// TIA Portal project "Fahrstuhl_V17" (V17)

(* hardware
DEVICE "S71500/ET200MP-Station_1"  S7-1500 station
   slot 0: "Profilschiene_0"  Rack  6ES7 590-1***0-0AA0
   slot 1: "SPS_Fahrstuhl"  CPU 1516F-3 PN/DP  6ES7 516-3FN01-0AB0  V2.9
      slot 3: "CPU-Display_1"  6ES7591-1BA00-0AA0
      slot 32768: "PROFINET-Schnittstelle_1"  X1
         slot 32769: "Port_1"  X1 P1
         slot 32770: "Port_2"  X1 P2
      slot 33024: "PROFINET-Schnittstelle_2"  X2
         slot 33025: "Port_1"  X2 P1
      slot 33280: "DP-Schnittstelle_1"  X3
      slot 34817: "Virtual CP interface port_1"  Virtual CP interface port  Virtual CP interface port
   slot 2: "DI 32x24VDC HF_1"  DI 32x24VDC HF  6ES7 521-1BL00-0AB0  V2.1
   slot 3: "DQ 32x24VDC/0.5A ST_1"  DQ 32x24VDC/0.5A ST  6ES7 522-1BL00-0AB0  V2.0
*)

// ===== PLC "SPS_Fahrstuhl"  CPU 1516F-3 PN/DP =====

VAR_GLOBAL   // PLC tag table "Standard-Variablentabelle"
   "Not-Aus" AT %I0.0 : Bool;   // Notausschalter Öffner
   "Automatikbetrieb" AT %I0.1 : Bool;   // Schalter Automatikbetrieb
   "Hand Hub Heben" AT %I0.2 : Bool;   // Schalter Kabine heben
   "Hand Hub Senken" AT %I0.3 : Bool;   // Schalter Kabine senken
   "Hand Tür auf" AT %I0.4 : Bool;   // Schalter Tür auf
   "Hand Tür zu" AT %I0.5 : Bool;   // Schalter Tür zu
   "Reserve_Eingang_0" AT %I0.6 : Bool;   // Reserve
   "Reserve_Eingang_1" AT %I0.7 : Bool;   // Reserve
   "Endlage zu tief" AT %I1.0 : Bool;   // Öffner
   "Endlage Etage I Halt" AT %I1.1 : Bool;   // Endlagenschalter Etage I Halt
   "Endlage Etage I Langsam" AT %I1.2 : Bool;   // Endlagenschalter Etage I Langsam
   "Endlage Etage II Halt" AT %I1.3 : Bool;   // Endlagenschalter Etage II Halt
   "Endlage Etage II Langsam" AT %I1.4 : Bool;   // Endlagenschalter Etage II Langsam
   "Endlage Etage III Halt" AT %I1.5 : Bool;   // Endlagenschalter Etage III Halt
   "Endlage Etage III Langsam" AT %I1.6 : Bool;   // Endlagenschalter Etage III Langsam
   "Endlage zu hoch" AT %I1.7 : Bool;   // Endlagenschalter zu hoch
   "Reserve_Eingang_2" AT %I2.0 : Bool;   // Reserve
   "Reserve_Eingang_3" AT %I2.1 : Bool;   // Reserve
   "Endlage Tür III Zu" AT %I2.2 : Bool;   // Endlagenschalter Tür III Zu
   "Endlage Tür III Auf" AT %I2.3 : Bool;   // Endlagenschalter Tür III Auf
   "Endlage Tür II Zu" AT %I2.4 : Bool;   // Endlagenschalter Tür II Zu
   "Endlage Tür II Auf" AT %I2.5 : Bool;   // Endlagenschalter Tür II Auf
   "Endlage Tür I Zu" AT %I2.6 : Bool;   // Endlagenschalter Tür I Zu
   "Endlage Tür I Auf" AT %I2.7 : Bool;   // Endlagenschalter Tür I Auf
   "Taster auf Etage III - Ab" AT %I3.0 : Bool;   // Taster auf Etage III - Ab
   "Taster auf Etage II - Ab" AT %I3.1 : Bool;   // Taster auf Etage II - Ab
   "Taster auf Etage II - Auf" AT %I3.2 : Bool;   // Taster auf Etage II - Auf
   "Taster auf Etage I - Auf" AT %I3.3 : Bool;   // Taster auf Etage I - Auf
   "Taster Lift nach III" AT %I3.4 : Bool;   // Taster Lift nach III
   "Taster Lift nach II" AT %I3.5 : Bool;   // Taster Lift nach II
   "Taster Lift nach I" AT %I3.6 : Bool;   // Taster Lift nach I
   "Reserve_Eingang_4" AT %I3.7 : Bool;   // Reserve
   "Hubmotor langsam Heben" AT %Q4.0 : Bool;   // Hubmotor langsam Heben
   "Hubmotor langsam Senken" AT %Q4.1 : Bool;   // Hubmotor langsam Senken
   "Hubmotor schnell Heben" AT %Q4.2 : Bool;   // Hubmotor schnell Heben
   "Hubmotor schnell Senken" AT %Q4.3 : Bool;   // Hubmotor schnell Senken
   "Türantrieb Etage I Öffnen" AT %Q4.4 : Bool;   // Türantrieb Etage I Öffnen
   "Türantrieb Etage I Schließen" AT %Q4.5 : Bool;   // Türantrieb Etage I Schließen
   "Türantrieb Etage II Öffnen" AT %Q4.6 : Bool;   // Türantrieb Etage II Öffnen
   "Türantrieb Etage II Schließen" AT %Q4.7 : Bool;   // Türantrieb Etage II Schließen
   "Türantrieb Etage III Öffnen" AT %Q5.0 : Bool;   // Türantrieb Etage III Öffnen
   "Türantrieb Etage III Schließen" AT %Q5.1 : Bool;   // Türantrieb Etage III Schließen
   "LED Lift nach I" AT %Q5.2 : Bool;   // LED Lift nach I
   "LED Lift nach II" AT %Q5.3 : Bool;   // LED Lift nach II
   "LED Lift nach III" AT %Q5.4 : Bool;   // LED Lift nach III
   "LED Etage I Lift Auf" AT %Q5.5 : Bool;   // LED Etage I Lift Auf
   "LED Etage II Lift Auf" AT %Q5.6 : Bool;   // LED Etage II Lift Auf
   "LED Etage II Lift Ab" AT %Q5.7 : Bool;   // LED Etage II Lift Ab
   "7-Segment G" AT %Q6.0 : Bool;   // 7-Segment G
   "7-Segment A" AT %Q6.1 : Bool;   // 7-Segment A
   "7-Segment B" AT %Q6.2 : Bool;   // 7-Segment B
   "7-Segment C" AT %Q6.3 : Bool;   // 7-Segment C
   "7-Segment D" AT %Q6.4 : Bool;   // 7-Segment D
   "7-Segment E" AT %Q6.5 : Bool;   // 7-Segment E
   "7-Segment F" AT %Q6.6 : Bool;   // 7-Segment F
   "LED Etage Lift III Ab" AT %Q6.7 : Bool;   // LED Etage Lift III Ab
   "Reserve_Ausgang_0" AT %Q7.0 : Bool;   // Reserve
   "Reserve_Ausgang_1" AT %Q7.1 : Bool;   // Reserve
   "Reserve_Ausgang_2" AT %Q7.2 : Bool;   // Reserve
   "Reserve_Ausgang_3" AT %Q7.3 : Bool;   // Reserve
   "Reserve_Ausgang_4" AT %Q7.4 : Bool;   // Reserve
   "Reserve_Ausgang_5" AT %Q7.5 : Bool;   // Reserve
   "Reserve_Ausgang_6" AT %Q7.6 : Bool;   // Reserve
   "Reserve_Ausgang_7" AT %Q7.7 : Bool;   // Reserve
   "Clock_Byte" AT %MB0 : Byte;
   "Clock_10Hz" AT %M0.0 : Bool;
   "Clock_5Hz" AT %M0.1 : Bool;
   "Clock_2.5Hz" AT %M0.2 : Bool;
   "Clock_2Hz" AT %M0.3 : Bool;
   "Clock_1.25Hz" AT %M0.4 : Bool;
   "Clock_1Hz" AT %M0.5 : Bool;
   "Clock_0.625Hz" AT %M0.6 : Bool;
   "Clock_0.5Hz" AT %M0.7 : Bool;
END_VAR

// folder: IDB's

DATA_BLOCK "Tür zu_DB"   // DB1
{ S7_Optimized_Access := 'TRUE' }
VERSION : 0.1
// stored: InstanceOfName Tür zu
"Tür zu"
BEGIN
END_DATA_BLOCK

DATA_BLOCK "Tür auf_DB"   // DB2
{ S7_Optimized_Access := 'TRUE' }
VERSION : 0.1
// stored: InstanceOfName Tür auf
"Tür auf"
BEGIN
END_DATA_BLOCK

DATA_BLOCK "Automatik_DB"   // DB3
{ S7_Optimized_Access := 'TRUE' }
VERSION : 0.1
// stored: InstanceOfName Automatik
"Automatik"
BEGIN
END_DATA_BLOCK

DATA_BLOCK "Hochfahren_DB"   // DB4
{ S7_Optimized_Access := 'TRUE' }
VERSION : 0.1
// stored: InstanceOfName Hochfahren
"Hochfahren"
BEGIN
END_DATA_BLOCK

DATA_BLOCK "Runterfahren_DB"   // DB5
{ S7_Optimized_Access := 'TRUE' }
VERSION : 0.1
// stored: InstanceOfName Runterfahren
"Runterfahren"
BEGIN
END_DATA_BLOCK

DATA_BLOCK "7-Segment Anzeige_DB"   // DB7
{ S7_Optimized_Access := 'TRUE' }
VERSION : 0.1
// stored: InstanceOfName 7-Segment Anzeige
"7-Segment Anzeige"
BEGIN
END_DATA_BLOCK

DATA_BLOCK "LED-Funktionen_DB"   // DB8
{ S7_Optimized_Access := 'TRUE' }
VERSION : 0.1
// stored: InstanceOfName LED-Funktionen
"LED-Funktionen"
BEGIN
END_DATA_BLOCK

DATA_BLOCK "Merker_DB"   // DB9
{ S7_Optimized_Access := 'TRUE' }
VERSION : 0.1
// stored: InstanceOfName Merker
"Merker"
BEGIN
END_DATA_BLOCK

DATA_BLOCK "Zeitbaustein Priorisierung_DB"   // DB12
{ S7_Optimized_Access := 'TRUE' }
VERSION : 0.1
// stored: InstanceOfName Zeitbaustein Priorisierung
"Zeitbaustein Priorisierung"
BEGIN
END_DATA_BLOCK

DATA_BLOCK "Handbetrieb_DB"   // DB13
{ S7_Optimized_Access := 'TRUE' }
VERSION : 0.1
// stored: InstanceOfName Handbetrieb
"Handbetrieb"
BEGIN
END_DATA_BLOCK

// folder: System blocks/Program resources

DATA_BLOCK "Timer Etage 1"   // DB10
{ S7_Optimized_Access := 'TRUE' }
AUTHOR : Simatic
FAMILY : IEC
NAME : IEC_TMR
VERSION : 1.0
// stored: InstanceOfName IEC_TIMER
"IEC_TIMER"
BEGIN
END_DATA_BLOCK

DATA_BLOCK "Timer Etage 3"   // DB11
{ S7_Optimized_Access := 'TRUE' }
AUTHOR : Simatic
FAMILY : IEC
NAME : IEC_TMR
VERSION : 1.0
// stored: InstanceOfName IEC_TIMER
"IEC_TIMER"
BEGIN
END_DATA_BLOCK

// folder: (top level)

ORGANIZATION_BLOCK "Main"   // OB1, FBD, ProgramCycle
TITLE = "Main Program Sweep (Cycle)"
{ S7_Optimized_Access := 'TRUE' }
VERSION : 0.1
// Belegung aller Ein- und Ausgänge  der FBs.
   VAR_INPUT
      Initial_Call : Bool;   // Initial call of this OB
      Remanence : Bool;   // =True, if remanent data are available
   END_VAR
   VAR_TEMP
      Automatikstart : Bool;
      "Not-Aus quittiert" : Bool;
   END_VAR
   VAR_TEMP   // added for the SCL form of the ladder/FBD networks
      _w1 : Bool;
      _w2 : Bool;
   END_VAR
BEGIN

REGION Network 1: Tür zu
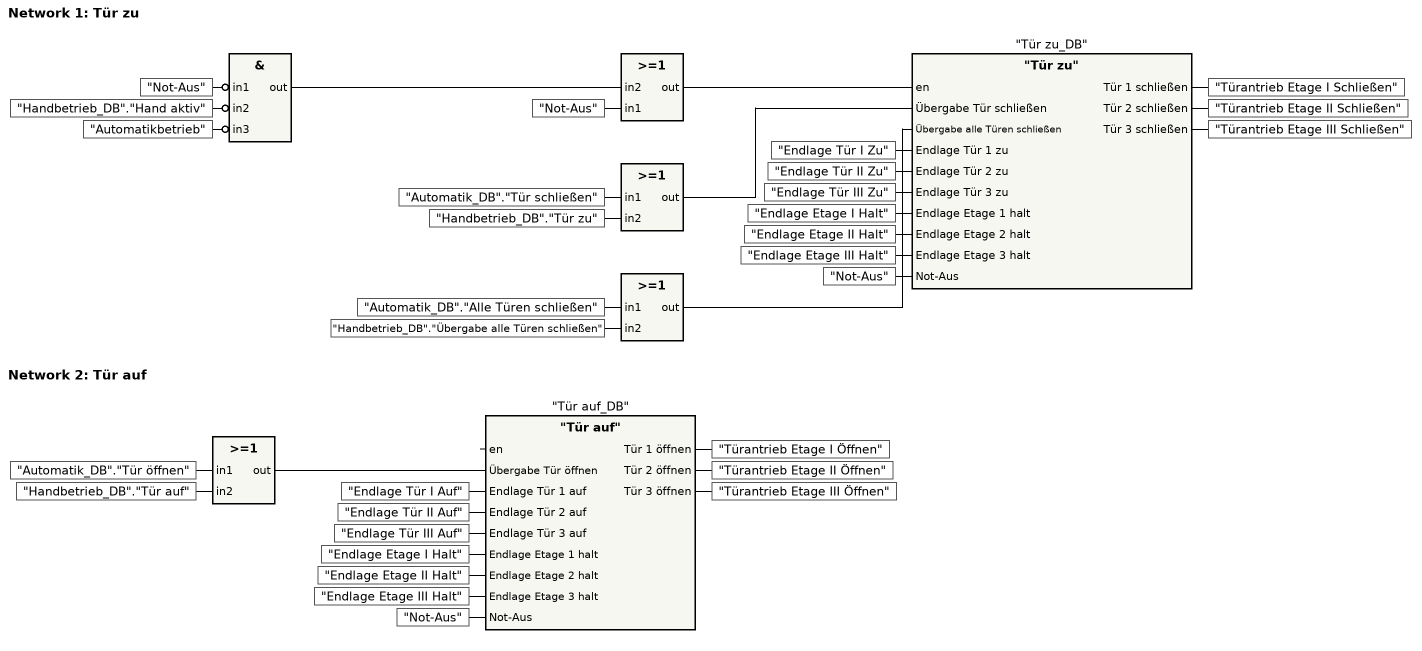
   IF (NOT "Not-Aus" AND NOT "Handbetrieb_DB"."Hand aktiv" AND NOT "Automatikbetrieb") OR "Not-Aus" THEN
       "Tür zu_DB"("Übergabe Tür schließen" := "Automatik_DB"."Tür schließen" OR "Handbetrieb_DB"."Tür zu",   // "Tür zu"
                   "Übergabe alle Türen schließen" := "Automatik_DB"."Alle Türen schließen" OR "Handbetrieb_DB"."Übergabe alle Türen schließen",
                   "Endlage Tür 1 zu" := "Endlage Tür I Zu",
                   "Endlage Tür 2 zu" := "Endlage Tür II Zu",
                   "Endlage Tür 3 zu" := "Endlage Tür III Zu",
                   "Endlage Etage 1 halt" := "Endlage Etage I Halt",
                   "Endlage Etage 2 halt" := "Endlage Etage II Halt",
                   "Endlage Etage 3 halt" := "Endlage Etage III Halt",
                   "Not-Aus" := "Not-Aus",
                   "Tür 1 schließen" => "Türantrieb Etage I Schließen",
                   "Tür 2 schließen" => "Türantrieb Etage II Schließen",
                   "Tür 3 schließen" => "Türantrieb Etage III Schließen");
   END_IF;
END_REGION

REGION Network 2: Tür auf
   "Tür auf_DB"("Übergabe Tür öffnen" := "Automatik_DB"."Tür öffnen" OR "Handbetrieb_DB"."Tür auf",   // "Tür auf"
                "Endlage Tür 1 auf" := "Endlage Tür I Auf",
                "Endlage Tür 2 auf" := "Endlage Tür II Auf",
                "Endlage Tür 3 auf" := "Endlage Tür III Auf",
                "Endlage Etage 1 halt" := "Endlage Etage I Halt",
                "Endlage Etage 2 halt" := "Endlage Etage II Halt",
                "Endlage Etage 3 halt" := "Endlage Etage III Halt",
                "Not-Aus" := "Not-Aus",
                "Tür 1 öffnen" => "Türantrieb Etage I Öffnen",
                "Tür 2 öffnen" => "Türantrieb Etage II Öffnen",
                "Tür 3 öffnen" => "Türantrieb Etage III Öffnen");
END_REGION

REGION Network 3: Automatik
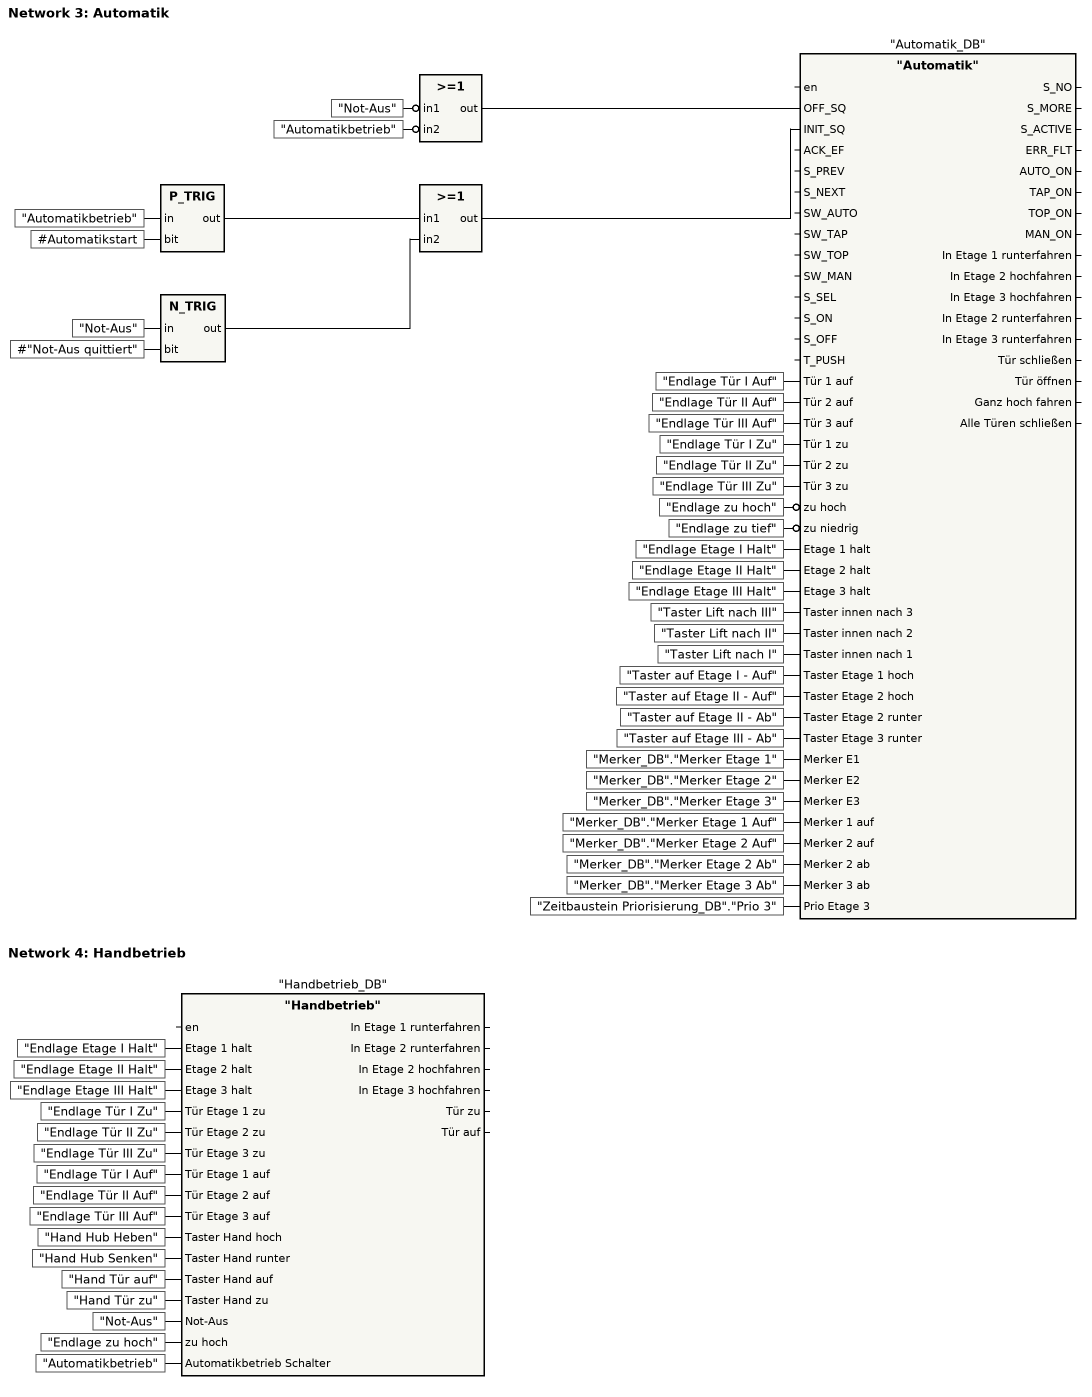
   #_w1 := "Automatikbetrieb" AND NOT #Automatikstart;   // rising edge
   #Automatikstart := "Automatikbetrieb";
   #_w2 := NOT "Not-Aus" AND #"Not-Aus quittiert";   // falling edge
   #"Not-Aus quittiert" := "Not-Aus";
   "Automatik_DB"(OFF_SQ := NOT "Not-Aus" OR NOT "Automatikbetrieb",   // "Automatik"
                  INIT_SQ := #_w1 OR #_w2,
                  "Tür 1 auf" := "Endlage Tür I Auf",
                  "Tür 2 auf" := "Endlage Tür II Auf",
                  "Tür 3 auf" := "Endlage Tür III Auf",
                  "Tür 1 zu" := "Endlage Tür I Zu",
                  "Tür 2 zu" := "Endlage Tür II Zu",
                  "Tür 3 zu" := "Endlage Tür III Zu",
                  "zu hoch" := NOT "Endlage zu hoch",
                  "zu niedrig" := NOT "Endlage zu tief",
                  "Etage 1 halt" := "Endlage Etage I Halt",
                  "Etage 2 halt" := "Endlage Etage II Halt",
                  "Etage 3 halt" := "Endlage Etage III Halt",
                  "Taster innen nach 3" := "Taster Lift nach III",
                  "Taster innen nach 2" := "Taster Lift nach II",
                  "Taster innen nach 1" := "Taster Lift nach I",
                  "Taster Etage 1 hoch" := "Taster auf Etage I - Auf",
                  "Taster Etage 2 hoch" := "Taster auf Etage II - Auf",
                  "Taster Etage 2 runter" := "Taster auf Etage II - Ab",
                  "Taster Etage 3 runter" := "Taster auf Etage III - Ab",
                  "Merker E1" := "Merker_DB"."Merker Etage 1",
                  "Merker E2" := "Merker_DB"."Merker Etage 2",
                  "Merker E3" := "Merker_DB"."Merker Etage 3",
                  "Merker 1 auf" := "Merker_DB"."Merker Etage 1 Auf",
                  "Merker 2 auf" := "Merker_DB"."Merker Etage 2 Auf",
                  "Merker 2 ab" := "Merker_DB"."Merker Etage 2 Ab",
                  "Merker 3 ab" := "Merker_DB"."Merker Etage 3 Ab",
                  "Prio Etage 3" := "Zeitbaustein Priorisierung_DB"."Prio 3");
END_REGION

REGION Network 4: Handbetrieb
   "Handbetrieb_DB"("Etage 1 halt" := "Endlage Etage I Halt",   // "Handbetrieb"
                    "Etage 2 halt" := "Endlage Etage II Halt",
                    "Etage 3 halt" := "Endlage Etage III Halt",
                    "Tür Etage 1 zu" := "Endlage Tür I Zu",
                    "Tür Etage 2 zu" := "Endlage Tür II Zu",
                    "Tür Etage 3 zu" := "Endlage Tür III Zu",
                    "Tür Etage 1 auf" := "Endlage Tür I Auf",
                    "Tür Etage 2 auf" := "Endlage Tür II Auf",
                    "Tür Etage 3 auf" := "Endlage Tür III Auf",
                    "Taster Hand hoch" := "Hand Hub Heben",
                    "Taster Hand runter" := "Hand Hub Senken",
                    "Taster Hand auf" := "Hand Tür auf",
                    "Taster Hand zu" := "Hand Tür zu",
                    "Not-Aus" := "Not-Aus",
                    "zu hoch" := "Endlage zu hoch",
                    "Automatikbetrieb Schalter" := "Automatikbetrieb");
END_REGION

REGION Network 5: Hochfahren
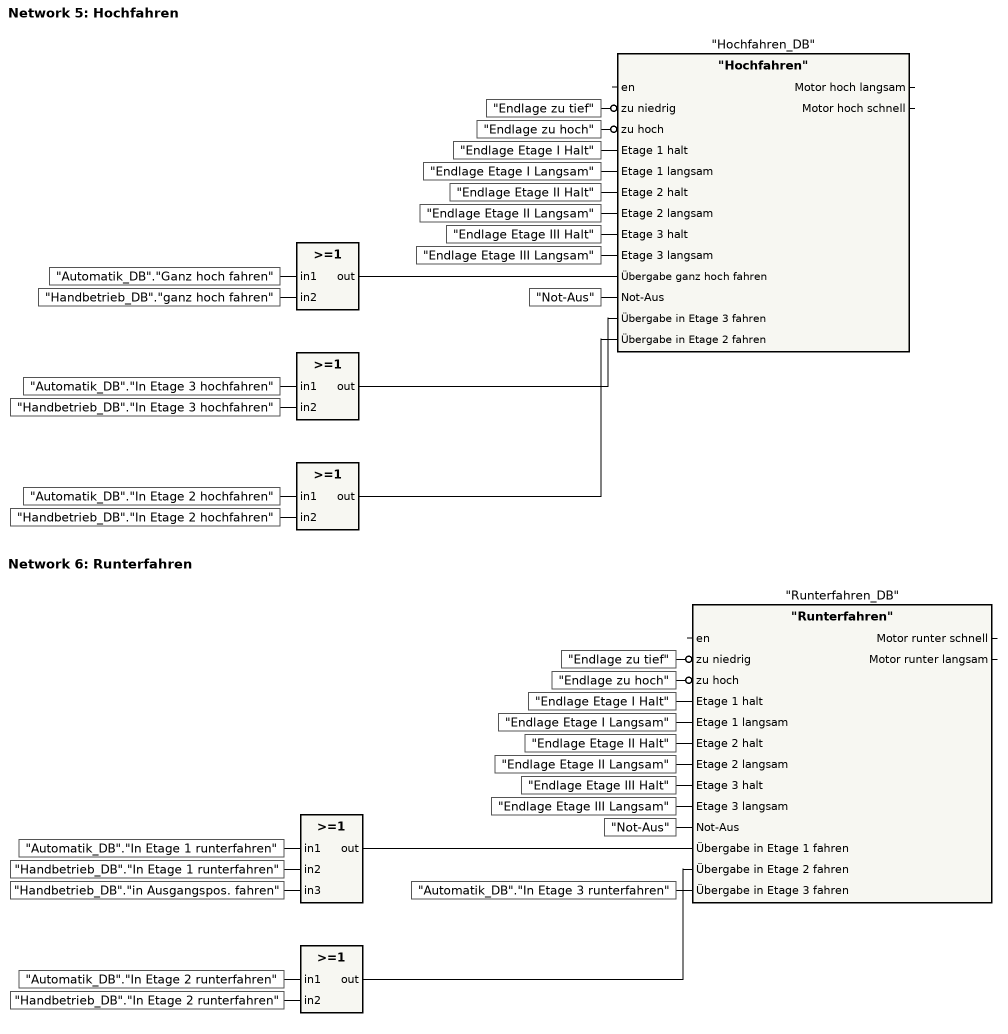
   "Hochfahren_DB"("zu niedrig" := NOT "Endlage zu tief",   // "Hochfahren"
                   "zu hoch" := NOT "Endlage zu hoch",
                   "Etage 1 halt" := "Endlage Etage I Halt",
                   "Etage 1 langsam" := "Endlage Etage I Langsam",
                   "Etage 2 halt" := "Endlage Etage II Halt",
                   "Etage 2 langsam" := "Endlage Etage II Langsam",
                   "Etage 3 halt" := "Endlage Etage III Halt",
                   "Etage 3 langsam" := "Endlage Etage III Langsam",
                   "Übergabe ganz hoch fahren" := "Automatik_DB"."Ganz hoch fahren" OR "Handbetrieb_DB"."ganz hoch fahren",
                   "Not-Aus" := "Not-Aus",
                   "Übergabe in Etage 3 fahren" := "Automatik_DB"."In Etage 3 hochfahren" OR "Handbetrieb_DB"."In Etage 3 hochfahren",
                   "Übergabe in Etage 2 fahren" := "Automatik_DB"."In Etage 2 hochfahren" OR "Handbetrieb_DB"."In Etage 2 hochfahren");
END_REGION

REGION Network 6: Runterfahren
   "Runterfahren_DB"("zu niedrig" := NOT "Endlage zu tief",   // "Runterfahren"
                     "zu hoch" := NOT "Endlage zu hoch",
                     "Etage 1 halt" := "Endlage Etage I Halt",
                     "Etage 1 langsam" := "Endlage Etage I Langsam",
                     "Etage 2 halt" := "Endlage Etage II Halt",
                     "Etage 2 langsam" := "Endlage Etage II Langsam",
                     "Etage 3 halt" := "Endlage Etage III Halt",
                     "Etage 3 langsam" := "Endlage Etage III Langsam",
                     "Not-Aus" := "Not-Aus",
                     "Übergabe in Etage 1 fahren" := "Automatik_DB"."In Etage 1 runterfahren" OR "Handbetrieb_DB"."In Etage 1 runterfahren" OR "Handbetrieb_DB"."in Ausgangspos. fahren",
                     "Übergabe in Etage 2 fahren" := "Automatik_DB"."In Etage 2 runterfahren" OR "Handbetrieb_DB"."In Etage 2 runterfahren",
                     "Übergabe in Etage 3 fahren" := "Automatik_DB"."In Etage 3 runterfahren");
END_REGION

REGION Network 7: Ausgänge Mehrfachbelegung
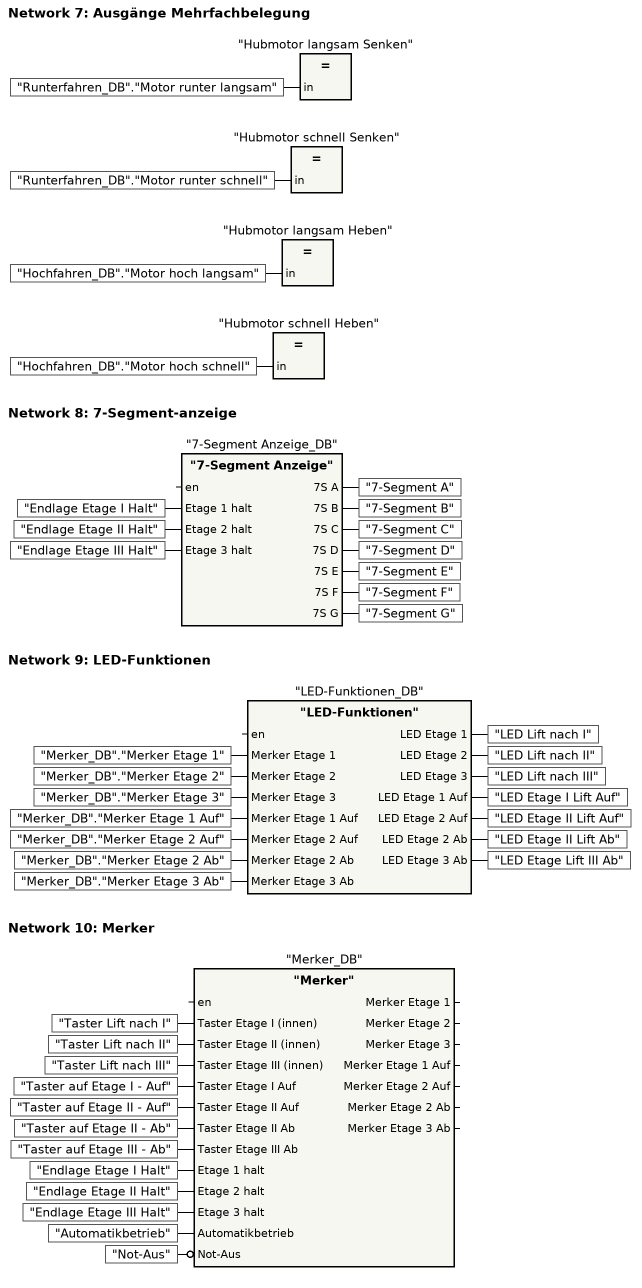
   "Hubmotor langsam Senken" := "Runterfahren_DB"."Motor runter langsam";
   "Hubmotor schnell Senken" := "Runterfahren_DB"."Motor runter schnell";
   "Hubmotor langsam Heben" := "Hochfahren_DB"."Motor hoch langsam";
   "Hubmotor schnell Heben" := "Hochfahren_DB"."Motor hoch schnell";
END_REGION

REGION Network 8: 7-Segment-anzeige
   "7-Segment Anzeige_DB"("Etage 1 halt" := "Endlage Etage I Halt",   // "7-Segment Anzeige"
                          "Etage 2 halt" := "Endlage Etage II Halt",
                          "Etage 3 halt" := "Endlage Etage III Halt",
                          "7S A" => "7-Segment A",
                          "7S B" => "7-Segment B",
                          "7S C" => "7-Segment C",
                          "7S D" => "7-Segment D",
                          "7S E" => "7-Segment E",
                          "7S F" => "7-Segment F",
                          "7S G" => "7-Segment G");
END_REGION

REGION Network 9: LED-Funktionen
   "LED-Funktionen_DB"("Merker Etage 1" := "Merker_DB"."Merker Etage 1",   // "LED-Funktionen"
                       "Merker Etage 2" := "Merker_DB"."Merker Etage 2",
                       "Merker Etage 3" := "Merker_DB"."Merker Etage 3",
                       "Merker Etage 1 Auf" := "Merker_DB"."Merker Etage 1 Auf",
                       "Merker Etage 2 Auf" := "Merker_DB"."Merker Etage 2 Auf",
                       "Merker Etage 2 Ab" := "Merker_DB"."Merker Etage 2 Ab",
                       "Merker Etage 3 Ab" := "Merker_DB"."Merker Etage 3 Ab",
                       "LED Etage 1" => "LED Lift nach I",
                       "LED Etage 2" => "LED Lift nach II",
                       "LED Etage 3" => "LED Lift nach III",
                       "LED Etage 1 Auf" => "LED Etage I Lift Auf",
                       "LED Etage 2 Auf" => "LED Etage II Lift Auf",
                       "LED Etage 2 Ab" => "LED Etage II Lift Ab",
                       "LED Etage 3 Ab" => "LED Etage Lift III Ab");
END_REGION

REGION Network 10: Merker
   "Merker_DB"("Taster Etage I (innen)" := "Taster Lift nach I",   // "Merker"
               "Taster Etage II (innen)" := "Taster Lift nach II",
               "Taster Etage III (innen)" := "Taster Lift nach III",
               "Taster Etage I Auf" := "Taster auf Etage I - Auf",
               "Taster Etage II Auf" := "Taster auf Etage II - Auf",
               "Taster Etage II Ab" := "Taster auf Etage II - Ab",
               "Taster Etage III Ab" := "Taster auf Etage III - Ab",
               "Etage 1 halt" := "Endlage Etage I Halt",
               "Etage 2 halt" := "Endlage Etage II Halt",
               "Etage 3 halt" := "Endlage Etage III Halt",
               Automatikbetrieb := "Automatikbetrieb",
               "Not-Aus" := NOT "Not-Aus");
END_REGION

REGION Network 11: Priorisierung Zeitbaustein
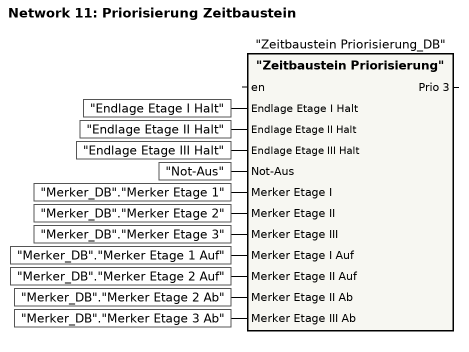
   "Zeitbaustein Priorisierung_DB"("Endlage Etage I Halt" := "Endlage Etage I Halt",   // "Zeitbaustein Priorisierung"
                           "Endlage Etage II Halt" := "Endlage Etage II Halt",
                           "Endlage Etage III Halt" := "Endlage Etage III Halt",
                           "Not-Aus" := "Not-Aus",
                           "Merker Etage I" := "Merker_DB"."Merker Etage 1",
                           "Merker Etage II" := "Merker_DB"."Merker Etage 2",
                           "Merker Etage III" := "Merker_DB"."Merker Etage 3",
                           "Merker Etage I Auf" := "Merker_DB"."Merker Etage 1 Auf",
                           "Merker Etage II Auf" := "Merker_DB"."Merker Etage 2 Auf",
                           "Merker Etage II Ab" := "Merker_DB"."Merker Etage 2 Ab",
                           "Merker Etage III Ab" := "Merker_DB"."Merker Etage 3 Ab");
END_REGION
END_ORGANIZATION_BLOCK

// folder: FB's

FUNCTION_BLOCK "Runterfahren"   // FB1, SCL
{ S7_Optimized_Access := 'TRUE' }
VERSION : 0.1
   VAR_INPUT
      "zu niedrig" : Bool;   // Endlage Fahrstuhl zu niedrig
      "zu hoch" : Bool;   // Endlage Fahrstuhl zu hoch
      "Etage 1 halt" : Bool;   // Endlage Etage 1
      "Etage 1 langsam" : Bool;   // Endlage Etage 1 langsamer
      "Etage 2 halt" : Bool;   // Endlage Etage 2
      "Etage 2 langsam" : Bool;   // Endlage Etage 2 langsamer
      "Etage 3 halt" : Bool;   // Endlage Etage 3
      "Etage 3 langsam" : Bool;   // Endlage Etage 3 langsamer
      "Not-Aus" : Bool;   // Notaus
      "Übergabe in Etage 1 fahren" : Bool;   // Fahrstuhl nach Etage 1
      "Übergabe in Etage 2 fahren" : Bool;   // Fahrstuhl nach Etage 2
      "Übergabe in Etage 3 fahren" : Bool;   // Fahrstuhl nach Etage 3
   END_VAR
   VAR_OUTPUT
      "Motor runter schnell" : Bool;   // Motoransteuerung langsam runter
      "Motor runter langsam" : Bool;   // Motoransteuerung schnell runter
   END_VAR
BEGIN
   (*Motor aus bei zu niedrig*)
   IF #"zu niedrig"=1 OR #"Not-Aus"=0 THEN
       #"Motor runter langsam" := 0;
       #"Motor runter schnell" := 0;
   END_IF;

   (*Ansteuerung bei Fahrt in Etage 3*)
   IF #"Übergabe in Etage 3 fahren"=1 AND #"Not-Aus"=1 THEN
       IF #"Etage 3 halt"=0 THEN
           #"Motor runter langsam" := 1;
       END_IF;
       IF #"Etage 3 halt" THEN
           #"Motor runter langsam":=0;
       END_IF;
   END_IF;

   (*Ansteuerung bei Fahrt in Etage 2*)
   IF #"Übergabe in Etage 2 fahren" = 1 AND #"Not-Aus" = 1 THEN
       IF #"Etage 2 halt" = 0 AND #"Etage 2 langsam" = 0 THEN
           #"Motor runter schnell" := 1;
       END_IF;
       IF #"Etage 2 halt" = 0 AND #"Etage 2 langsam" = 1 THEN
           #"Motor runter langsam" := 1;
           #"Motor runter schnell" := 0;
       END_IF;
       IF #"Etage 2 halt" = 1 THEN
           #"Motor runter langsam" := 0;
           #"Motor runter schnell" := 0;
       END_IF;
   END_IF;

   (*Ansteuerung bei Fahrt in Etage 1*)
   IF #"Übergabe in Etage 1 fahren" = 1 AND #"Not-Aus" = 1 THEN
       IF #"Etage 1 halt" = 0 AND #"Etage 1 langsam" = 0 THEN
           #"Motor runter schnell" := 1;
       END_IF;
       IF #"Etage 1 halt" = 0 AND #"Etage 1 langsam" = 1 THEN
           #"Motor runter langsam" := 1;
           #"Motor runter schnell" := 0;
       END_IF;
       IF #"Etage 1 halt" = 1 THEN
           #"Motor runter langsam" := 0;
           #"Motor runter schnell" := 0;
       END_IF;
   END_IF;

   (*Motor aus bei Betriebsartenänderung*)
   IF "Handbetrieb_DB"."Automatik neg. Flanke" OR "Handbetrieb_DB"."Handbetrieb neg. Flanke" THEN
       #"Motor runter langsam" := 0;
       #"Motor runter schnell" := 0;
   END_IF;
END_FUNCTION_BLOCK

FUNCTION_BLOCK "Hochfahren"   // FB2, SCL
{ S7_Optimized_Access := 'TRUE' }
VERSION : 0.1
   VAR_INPUT
      "zu niedrig" : Bool;   // Endlage Fahrstuhl zu niedrig
      "zu hoch" : Bool;   // Endlage Fahrstuhl zu hoch
      "Etage 1 halt" : Bool;   // Endlage Etage 1
      "Etage 1 langsam" : Bool;   // Endlage Etage 1 langsamer
      "Etage 2 halt" : Bool;   // Endlage Etage 2
      "Etage 2 langsam" : Bool;   // Endlage Etage 2 langsamer
      "Etage 3 halt" : Bool;   // Endlage Etage 3
      "Etage 3 langsam" : Bool;   // Endlage Etage 3 langsamer
      "Übergabe ganz hoch fahren" : Bool;   // Fahrstuhl ganz hoch
      "Not-Aus" : Bool;   // Notaus
      "Übergabe in Etage 3 fahren" : Bool;   // Fahrstuhl nach Etage 3
      "Übergabe in Etage 2 fahren" : Bool;   // Fahrstuhl nach Etage 2
   END_VAR
   VAR_OUTPUT
      "Motor hoch langsam" : Bool;   // Motoransteuerung langsam hoch
      "Motor hoch schnell" : Bool;   // Motoransteuerung schnell hoch
   END_VAR
BEGIN
   (*Motor aus bei zu hoch*)
   IF #"zu hoch"=1 OR #"Not-Aus"=0 THEN
       #"Motor hoch langsam" := 0;
       #"Motor hoch schnell":=0;
   END_IF;

   (*Ansteuerung ganz hoch*)
   IF #"Übergabe ganz hoch fahren" = 1 AND #"zu hoch" = 0 THEN
       #"Motor hoch schnell" := 1;
   END_IF;

   (*Ansteuerung bei Fahrt in Etage 3*)
   IF #"Übergabe in Etage 3 fahren" = 1 AND #"Not-Aus" = 1 THEN
       IF #"Etage 3 halt" = 0 AND #"Etage 3 langsam" = 0 THEN
           #"Motor hoch schnell" := 1;
       END_IF;
       IF #"Etage 3 halt" = 0 AND #"Etage 3 langsam" = 1 THEN
           #"Motor hoch langsam" := 1;
           #"Motor hoch schnell" := 0;
       END_IF;
       IF #"Etage 3 halt" = 1 THEN
           #"Motor hoch langsam" := 0;
           #"Motor hoch schnell" := 0;
       END_IF;
   END_IF;

   (*Ansteuerung bei Fahrt in Etage 2*)
   IF #"Übergabe in Etage 2 fahren" AND #"Not-Aus" = 1 THEN
       IF #"Etage 2 halt" = 0 AND #"Etage 2 langsam" = 0 THEN
           #"Motor hoch schnell" := 1;
       END_IF;
       IF #"Etage 2 halt" = 0 AND #"Etage 2 langsam" = 1 THEN
           #"Motor hoch langsam" := 1;
           #"Motor hoch schnell" := 0;
       END_IF;
       IF #"Etage 2 halt" = 1 THEN
           #"Motor hoch langsam" := 0;
           #"Motor hoch schnell" := 0;
       END_IF;
   END_IF;

   (*Motor aus bei Betriebsartenänderung*)
   IF  "Handbetrieb_DB"."Automatik neg. Flanke" THEN
       #"Motor hoch langsam" := 0;
       #"Motor hoch schnell" := 0;
   END_IF;
END_FUNCTION_BLOCK

FUNCTION_BLOCK "Tür auf"   // FB4, SCL
{ S7_Optimized_Access := 'TRUE' }
VERSION : 0.1
   VAR_INPUT
      "Übergabe Tür öffnen" : Bool;   // Übergabebit Tür öffnen
      "Endlage Tür 1 auf" : Bool;   // Endlage Tür 1 auf
      "Endlage Tür 2 auf" : Bool;   // Endlage Tür 2 auf
      "Endlage Tür 3 auf" : Bool;   // Endlage Tür 3 auf
      "Endlage Etage 1 halt" : Bool;   // Endlage Etage 1 halt
      "Endlage Etage 2 halt" : Bool;   // Endlage Etage 2 halt
      "Endlage Etage 3 halt" : Bool;   // Endlage Etage 3 halt
      "Not-Aus" : Bool;   // Notaus
   END_VAR
   VAR_OUTPUT
      "Tür 1 öffnen" : Bool;   // Befehl Tür 1 öffen
      "Tür 2 öffnen" : Bool;   // Befehl Tür 2 öffen
      "Tür 3 öffnen" : Bool;   // Befehl Tür 3 öffen
   END_VAR
BEGIN
   (*Tür 1*)
   IF #"Endlage Etage 1 halt" = 1 AND #"Endlage Tür 1 auf" = 0 AND #"Übergabe Tür öffnen" THEN
       #"Tür 1 öffnen" := 1
       ;
   END_IF;
   IF #"Endlage Tür 1 auf" = 1 OR #"Not-Aus" = 0 OR "Handbetrieb_DB"."Handbetrieb neg. Flanke" THEN
       #"Tür 1 öffnen" := 0
       ;
   END_IF;

   (*Tür 2*)
   IF #"Endlage Etage 2 halt" = 1 AND #"Endlage Tür 2 auf" = 0 AND #"Übergabe Tür öffnen" THEN
       #"Tür 2 öffnen" := 1
       ;
   END_IF;
   IF #"Endlage Tür 2 auf" = 1 OR #"Not-Aus"= 0  OR "Handbetrieb_DB"."Handbetrieb neg. Flanke" THEN
       #"Tür 2 öffnen" := 0
       ;
   END_IF;

   (*Tür 3*)
   IF #"Endlage Etage 3 halt" = 1 AND #"Endlage Tür 3 auf" = 0 AND #"Übergabe Tür öffnen" THEN
       #"Tür 3 öffnen" := 1
       ;
   END_IF;
   IF #"Endlage Tür 3 auf" = 1 OR #"Not-Aus" = 0 OR "Handbetrieb_DB"."Handbetrieb neg. Flanke" THEN
       #"Tür 3 öffnen" := 0
       ;
   END_IF;
END_FUNCTION_BLOCK

FUNCTION_BLOCK "Tür zu"   // FB5, SCL
{ S7_Optimized_Access := 'TRUE' }
VERSION : 0.1
   VAR_INPUT
      "Übergabe Tür schließen" : Bool;   // Übergabebit Tür schließen
      "Übergabe alle Türen schließen" : Bool;   // Übergabebit alle Türen schließen
      "Endlage Tür 1 zu" : Bool;   // Endlage Tür 1 zu
      "Endlage Tür 2 zu" : Bool;   // Endlage Tür 2 zu
      "Endlage Tür 3 zu" : Bool;   // Endlage Tür 3 zu
      "Endlage Etage 1 halt" : Bool;   // Endlage Etage 1 halt
      "Endlage Etage 2 halt" : Bool;   // Endlage Etage 2 halt
      "Endlage Etage 3 halt" : Bool;   // Endlage Etage 3 halt
      "Not-Aus" : Bool;   // Notaus
   END_VAR
   VAR_OUTPUT
      "Tür 1 schließen" : Bool;   // Befehl Tür 1 schließen
      "Tür 2 schließen" : Bool;   // Befehl Tür 2 schließen
      "Tür 3 schließen" : Bool;   // Befehl Tür 3 schließen
   END_VAR
BEGIN
   (*Tür 1*)
   IF #"Endlage Etage 1 halt" AND #"Endlage Tür 1 zu" = 0 AND #"Übergabe Tür schließen" OR #"Übergabe alle Türen schließen" THEN
       #"Tür 1 schließen" := 1
       ;
   END_IF;
   IF #"Endlage Tür 1 zu" OR #"Not-Aus" = 0 THEN
       #"Tür 1 schließen" := 0
       ;
   END_IF;

   (*Tür 2*)
   IF #"Endlage Etage 2 halt" AND #"Endlage Tür 2 zu" = 0 AND #"Übergabe Tür schließen" OR #"Übergabe alle Türen schließen" THEN
       #"Tür 2 schließen" := 1
       ;
   END_IF;
   IF #"Endlage Tür 2 zu" OR #"Not-Aus" = 0 THEN
       #"Tür 2 schließen" := 0
       ;
   END_IF;

   (*Tür 3*)
   IF #"Endlage Etage 3 halt" AND #"Endlage Tür 3 zu" = 0 AND #"Übergabe Tür schließen" OR #"Übergabe alle Türen schließen" THEN
       #"Tür 3 schließen" := 1
       ;
   END_IF;
   IF #"Endlage Tür 3 zu" OR #"Not-Aus" = 0 THEN
       #"Tür 3 schließen" := 0
       ;
   END_IF;
END_FUNCTION_BLOCK

FUNCTION_BLOCK "Automatik"   // FB6, GRAPH_PLUS
{ S7_Optimized_Access := 'TRUE' }
VERSION : 0.1
   VAR_INPUT
      OFF_SQ : Bool := false;   // Kette ausschalten
      INIT_SQ : Bool := false;   // Kette in Initialzustand versetzen
      ACK_EF : Bool := false;   // Alle Fehler und Störungen quittieren
      S_PREV : Bool := false;   // Vorherigen Schritt am Parameter S_NO ausgeben
      S_NEXT : Bool := false;   // Nächsten Schritt am Parameter S_NO anzeigen
      SW_AUTO : Bool := false;   // Automatischer Betrieb
      SW_TAP : Bool := false;   // Halbautomatisch/Weiterschalten mit Transition
      SW_TOP : Bool := false;   // Halbautomatisch/Ignoriere Transition
      SW_MAN : Bool := false;   // Handbetrieb
      S_SEL : Int := 0;   // Schritt auswählen, der an S_NO ausgegeben werden soll
      S_ON : Bool := false;   // Schritt aktivieren, der an Parameter S_NO anliegt
      S_OFF : Bool := false;   // Schritt deaktivieren, der an Parameter S_NO anliegt
      T_PUSH : Bool := false;   // Schaltfreigabe für Transition im halbautomatischen Betrieb
      "Tür 1 auf" : Bool;   // Endlage Tür 1 auf
      "Tür 2 auf" : Bool;   // Endlage Tür 2 auf
      "Tür 3 auf" : Bool;   // Endlage Tür 3 auf
      "Tür 1 zu" : Bool;   // Endlage Tür 1 zu
      "Tür 2 zu" : Bool;   // Endlage Tür 2 zu
      "Tür 3 zu" : Bool;   // Endlage Tür 3 zu
      "zu hoch" : Bool;   // Endlage Fahrstuhl zu hoch
      "zu niedrig" : Bool;   // Endlage Fahrstuhl zu niedrig
      "Etage 1 halt" : Bool;   // Endlage Etage 1
      "Etage 2 halt" : Bool;   // Endlage Etage 2
      "Etage 3 halt" : Bool;   // Endlage Etage 3
      "Taster innen nach 3" : Bool;   // Taster innen nach Etage 3
      "Taster innen nach 2" : Bool;   // Taster innen nach Etage 2
      "Taster innen nach 1" : Bool;   // Taster innen nach Etage 1
      "Taster Etage 1 hoch" : Bool;   // Taster aus Etage 1 hoch
      "Taster Etage 2 hoch" : Bool;   // Taster aus Etage 2 hoch
      "Taster Etage 2 runter" : Bool;   // Taster aus Etage 2 runter
      "Taster Etage 3 runter" : Bool;   // Taster aus Etage 3 runter
      "Merker E1" : Bool;   // Anforderung Etage 1 innen
      "Merker E2" : Bool;   // Anforderung Etage 2 innen
      "Merker E3" : Bool;   // Anforderung Etage 3 innen
      "Merker 1 auf" : Bool;   // Anforderung Etage 1 hoch
      "Merker 2 auf" : Bool;   // Anforderung Etage 2 hoch
      "Merker 2 ab" : Bool;   // Anforderung Etage 2 runter
      "Merker 3 ab" : Bool;   // Anforderung Etage 3 runter
      "Prio Etage 3" : Bool;   // Priorisierung Etage 3
   END_VAR
   VAR_OUTPUT
      S_NO : Int := 0;   // Schrittnummer
      S_MORE : Bool := false;   // Weitere Schritte sind vorhanden und können in S_NO angezeigt werden.
      S_ACTIVE : Bool := false;   // Schritt, der an Parameter S_NO angezeigt wird, ist aktiv
      ERR_FLT : Bool := false;   // Sammelfehler Interlock oder Supervision
      AUTO_ON : Bool := false;   // Automatischer Betrieb eingeschaltet
      TAP_ON : Bool := false;   // Halbautomatischer Betrieb/Schritt mit Transition eingeschaltet
      TOP_ON : Bool := false;   // Halbautomatischer Betrieb/Ignoriere Transition eingeschaltet
      MAN_ON : Bool := false;   // Handbetrieb eingeschaltet
      "In Etage 1 runterfahren" : Bool;   // Fahrbefehl in Etage 1 runter
      "In Etage 2 hochfahren" : Bool;   // Fahrbefehl in Etage 2 hoch
      "In Etage 3 hochfahren" : Bool;   // Fahrbefehl in Etage 3 hoch
      "In Etage 2 runterfahren" : Bool;   // Fahrbefehl in Etage 2 runter
      "In Etage 3 runterfahren" : Bool;   // Fahrbefehl in Etage 3 runter
      "Tür schließen" : Bool;   // Befehl Tür schließen
      "Tür öffnen" : Bool;   // Befehl Tür öffnen
      "Ganz hoch fahren" : Bool;   // Fahrstuhl an oberste Endlage
      "Alle Türen schließen" : Bool;   // Befehl alle Türen zu
   END_VAR
   VAR
      richten : Bool;   // Richtbetrieb
      HMI_INFO : Array[0..8] of UInt;
      IF_PAR : G7_IfParPlus_V2;
      RT_DATA : G7_RTDataPlus_V2;   // Interner Datenbereich
      "alle Türen zu" : G7_TransitionPlus_V2;   // Transitionsstruktur
      "ganz oben" : G7_TransitionPlus_V2;   // Transitionsstruktur
      Gerichtet : G7_TransitionPlus_V2;   // Transitionsstruktur
      "T: 1 nach 2" : G7_TransitionPlus_V2;   // Transitionsstruktur
      "Etage 2 halt #2" : G7_TransitionPlus_V2;   // Transitionsstruktur
      "Tür auf Etage 2 #2" : G7_TransitionPlus_V2;   // Transitionsstruktur
      "Tür zu Etage 2 #2" : G7_TransitionPlus_V2;   // Transitionsstruktur
      "T: 2 nach 1" : G7_TransitionPlus_V2;   // Transitionsstruktur
      "Etage 1 halt #2" : G7_TransitionPlus_V2;   // Transitionsstruktur
      "Tür auf Etage 1 #3" : G7_TransitionPlus_V2;   // Transitionsstruktur
      "Tür zu Etage 1 #3" : G7_TransitionPlus_V2;   // Transitionsstruktur
      "T: 2 nach 3" : G7_TransitionPlus_V2;   // Transitionsstruktur
      "Etage 3 halt #2" : G7_TransitionPlus_V2;   // Transitionsstruktur
      "Tür auf Etage 3 #3" : G7_TransitionPlus_V2;   // Transitionsstruktur
      "Tür zu Etage 3 #3" : G7_TransitionPlus_V2;   // Transitionsstruktur
      "In 2 bleiben" : G7_TransitionPlus_V2;   // Transitionsstruktur
      "Tür auf Etage 2 #3" : G7_TransitionPlus_V2;   // Transitionsstruktur
      "Tür zu Etage 2 #3" : G7_TransitionPlus_V2;   // Transitionsstruktur
      "T: 1 nach 3" : G7_TransitionPlus_V2;   // Transitionsstruktur
      "Etage 3 halt #1" : G7_TransitionPlus_V2;   // Transitionsstruktur
      "Tür auf Etage 3 #1" : G7_TransitionPlus_V2;   // Transitionsstruktur
      "Tür zu Etage 3 #1" : G7_TransitionPlus_V2;   // Transitionsstruktur
      "T: 3 nach 2" : G7_TransitionPlus_V2;   // Transitionsstruktur
      "Etage 2 halt #1" : G7_TransitionPlus_V2;   // Transitionsstruktur
      "Tür auf Etage 2 #1" : G7_TransitionPlus_V2;   // Transitionsstruktur
      "Tür zu Etage 2 #1" : G7_TransitionPlus_V2;   // Transitionsstruktur
      "T: 3 nach 1" : G7_TransitionPlus_V2;   // Transitionsstruktur
      "Etage 1 halt #1" : G7_TransitionPlus_V2;   // Transitionsstruktur
      "Tür auf Etage 1 #1" : G7_TransitionPlus_V2;   // Transitionsstruktur
      "Tür zu Etage 1 #1" : G7_TransitionPlus_V2;   // Transitionsstruktur
      "In 3 bleiben" : G7_TransitionPlus_V2;   // Transitionsstruktur
      "Tür auf Etage 3 #2" : G7_TransitionPlus_V2;   // Transitionsstruktur
      "Tür zu Etage 3 #2" : G7_TransitionPlus_V2;   // Transitionsstruktur
      "In 1 bleiben" : G7_TransitionPlus_V2;   // Transitionsstruktur
      "Tür auf Etage 1 #2" : G7_TransitionPlus_V2;   // Transitionsstruktur
      "Tür zu Etage 1 #2" : G7_TransitionPlus_V2;   // Transitionsstruktur
      Trans37 : G7_TransitionPlus_V2;   // Transitionsstruktur
      Trans38 : G7_TransitionPlus_V2;   // Transitionsstruktur
      Startschritt : G7_StepPlus_V2;   // Schrittstruktur
      "Start: 2" : G7_StepPlus_V2;   // Schrittstruktur
      "Start: 3" : G7_StepPlus_V2;   // Schrittstruktur
      "warten in 1" : G7_StepPlus_V2;   // Schrittstruktur
      "1 nach 2" : G7_StepPlus_V2;   // Schrittstruktur
      "Tür auf in 2 #2" : G7_StepPlus_V2;   // Schrittstruktur
      "Tür zu in 2 #2" : G7_StepPlus_V2;   // Schrittstruktur
      "warten in 2" : G7_StepPlus_V2;   // Schrittstruktur
      "2 nach 1" : G7_StepPlus_V2;   // Schrittstruktur
      "Tür auf in 1 #3" : G7_StepPlus_V2;   // Schrittstruktur
      "Tür zu in 1 #3" : G7_StepPlus_V2;   // Schrittstruktur
      "2 nach 3" : G7_StepPlus_V2;   // Schrittstruktur
      "Tür auf in 3 #3" : G7_StepPlus_V2;   // Schrittstruktur
      "Tür zu in 3 #3" : G7_StepPlus_V2;   // Schrittstruktur
      "Tür auf in 2 #3" : G7_StepPlus_V2;   // Schrittstruktur
      "Tür zu in 2 #3" : G7_StepPlus_V2;   // Schrittstruktur
      "1 nach 3" : G7_StepPlus_V2;   // Schrittstruktur
      "Tür auf in 3 #1" : G7_StepPlus_V2;   // Schrittstruktur
      "Tür zu in 3 #1" : G7_StepPlus_V2;   // Schrittstruktur
      "warten in 3" : G7_StepPlus_V2;   // Schrittstruktur
      "3 nach 2" : G7_StepPlus_V2;   // Schrittstruktur
      "Tür auf in 2 #1" : G7_StepPlus_V2;   // Schrittstruktur
      "Tür zu in 2 #1" : G7_StepPlus_V2;   // Schrittstruktur
      "3 nach 1" : G7_StepPlus_V2;   // Schrittstruktur
      "Tür auf in 1 #1" : G7_StepPlus_V2;   // Schrittstruktur
      "Tür zu in 1 #1" : G7_StepPlus_V2;   // Schrittstruktur
      "Tür auf in 3 #2" : G7_StepPlus_V2;   // Schrittstruktur
      "Tür zu in 3 #2" : G7_StepPlus_V2;   // Schrittstruktur
      "Tür auf in 1 #2" : G7_StepPlus_V2;   // Schrittstruktur
      "Tür zu in 1 #2" : G7_StepPlus_V2;   // Schrittstruktur
      SINI : Array[0..1] of USInt;
      LSTT : Array[0..37] of USInt;
      ATAJ : Array[0..37] of USInt;
      ATAB : Array[0..37] of USInt;
      PSTT : Array[0..37] of USInt;
      NSTT : Array[0..37] of USInt;
      ASSJ : Array[0..29] of USInt;
      ASSB : Array[0..29] of USInt;
      PTTS : Array[0..29] of USInt;
      NTTS : Array[0..29] of USInt;
      SW_SQTS : Array[0..29] of USInt;
      SWITCH : Array[0..17] of USInt;
      TVX : Array[0..14] of USInt;
      TTX : Array[0..14] of USInt;
      TSX : Array[0..1] of USInt;
      S00X : Array[0..1] of USInt;
      SOFFX : Array[0..1] of USInt;
      SONX : Array[0..1] of USInt;
      SAX : Array[0..1] of USInt;
      SERRX : Array[0..30] of USInt;
      SMX : Array[0..30] of USInt;
      S0X : Array[0..30] of USInt;
      S1X : Array[0..30] of USInt;
      IL_ALARM_INST : Program_Alarm;
      SUP_ALARM_INST : Program_Alarm;
      STEP_TIME_ALARM_INST : Program_Alarm;
      IEC_TIMER_INST : IEC_TIMER;
      TRANSACTION_FLAG : Bool := false;
   END_VAR
   // SINI[0] := 2;
   // LSTT[0] := 255;
   // LSTT[1] := 255;
   // LSTT[2] := 255;
   // LSTT[3] := 255;
   // LSTT[4] := 255;
   // LSTT[5] := 255;
   // LSTT[6] := 255;
   // ATAJ[1] := 1;
   // ATAJ[2] := 2;
   // ATAJ[3] := 3;
   // ATAJ[4] := 4;
   // ATAJ[5] := 5;
   // ATAJ[6] := 6;
   // ATAB[1] := 1;
   // ATAB[2] := 2;
   // ATAB[3] := 33;
   // ATAB[4] := 4;
   // ATAB[5] := 5;
   // ATAB[6] := 6;
   // PSTT[1] := 1;
   // PSTT[2] := 2;
   // PSTT[3] := 3;
   // PSTT[4] := 4;
   // PSTT[5] := 5;
   // PSTT[6] := 6;
   // NSTT[0] := 1;
   // NSTT[1] := 2;
   // NSTT[2] := 3;
   // NSTT[3] := 4;
   // NSTT[4] := 5;
   // NSTT[5] := 6;
   // NSTT[6] := 7;
   // ASSJ[1] := 1;
   // ASSJ[2] := 2;
   // ASSJ[3] := 3;
   // ASSJ[4] := 4;
   // ASSJ[5] := 5;
   // ASSJ[6] := 6;
   // ASSB[1] := 1;
   // ASSB[2] := 2;
   // ASSB[3] := 3;
   // ASSB[4] := 4;
   // ASSB[5] := 5;
   // ASSB[6] := 6;
   // PTTS[0] := 255;
   // PTTS[2] := 1;
   // PTTS[3] := 2;
   // PTTS[4] := 3;
   // PTTS[5] := 4;
   // PTTS[6] := 5;
   // NTTS[1] := 1;
   // NTTS[2] := 2;
   // NTTS[3] := 18;
   // NTTS[4] := 4;
   // NTTS[5] := 5;
   // NTTS[6] := 6;
   // TVX[0] := 16#1;
   // TTX[0] := 16#1;
   // TSX[0] := 16#1;
   // S00X[0] := 16#1;
   // SOFFX[0] := 16#1;
   // SONX[0] := 16#1;
   // SAX[0] := 16#1;
   // SERRX[0] := 16#1;
   // SMX[0] := 16#1;
   // S0X[0] := 16#1;
   // S1X[0] := 16#1;
   // LSTT[7] := 255;
   // LSTT[8] := 255;
   // LSTT[9] := 255;
   // LSTT[10] := 3;
   // LSTT[11] := 255;
   // LSTT[12] := 255;
   // LSTT[13] := 255;
   // LSTT[14] := 19;
   // LSTT[15] := 255;
   // LSTT[16] := 255;
   // LSTT[17] := 7;
   // LSTT[18] := 255;
   // LSTT[19] := 255;
   // LSTT[20] := 255;
   // LSTT[21] := 255;
   // LSTT[22] := 255;
   // LSTT[23] := 255;
   // LSTT[24] := 255;
   // LSTT[25] := 7;
   // LSTT[26] := 255;
   // LSTT[27] := 255;
   // LSTT[28] := 255;
   // LSTT[29] := 3;
   // LSTT[30] := 255;
   // LSTT[31] := 255;
   // LSTT[32] := 19;
   // LSTT[33] := 255;
   // LSTT[34] := 255;
   // LSTT[35] := 3;
   // ATAJ[7] := 7;
   // ATAJ[8] := 8;
   // ATAJ[9] := 9;
   // ATAJ[10] := 10;
   // ATAJ[11] := 11;
   // ATAJ[12] := 12;
   // ATAJ[13] := 13;
   // ATAJ[14] := 14;
   // ATAJ[15] := 15;
   // ATAJ[16] := 16;
   // ATAJ[17] := 17;
   // ATAJ[18] := 18;
   // ATAJ[19] := 19;
   // ATAJ[20] := 20;
   // ATAJ[21] := 21;
   // ATAJ[22] := 22;
   // ATAJ[23] := 23;
   // ATAJ[24] := 24;
   // ATAJ[25] := 25;
   // ATAJ[26] := 26;
   // ATAJ[27] := 27;
   // ATAJ[28] := 28;
   // ATAJ[29] := 29;
   // ATAJ[30] := 30;
   // ATAJ[31] := 31;
   // ATAJ[32] := 32;
   // ATAJ[33] := 33;
   // ATAJ[34] := 34;
   // ATAJ[35] := 35;
   // ATAB[7] := 11;
   // ATAB[8] := 8;
   // ATAB[9] := 9;
   // ATAB[10] := 10;
   // ATAB[11] := 15;
   // ATAB[12] := 12;
   // ATAB[13] := 13;
   // ATAB[14] := 14;
   // ATAB[15] := 7;
   // ATAB[16] := 16;
   // ATAB[17] := 17;
   // ATAB[18] := 3;
   // ATAB[19] := 36;
   // ATAB[20] := 20;
   // ATAB[21] := 21;
   // ATAB[22] := 26;
   // ATAB[23] := 23;
   // ATAB[24] := 24;
   // ATAB[25] := 25;
   // ATAB[26] := 30;
   // ATAB[27] := 37;
   // ATAB[28] := 28;
   // ATAB[29] := 29;
   // ATAB[30] := 22;
   // ATAB[31] := 31;
   // ATAB[32] := 32;
   // ATAB[33] := 18;
   // ATAB[34] := 34;
   // ATAB[35] := 35;
   // PSTT[7] := 7;
   // PSTT[8] := 8;
   // PSTT[9] := 9;
   // PSTT[10] := 10;
   // PSTT[11] := 7;
   // PSTT[12] := 11;
   // PSTT[13] := 12;
   // PSTT[14] := 13;
   // PSTT[15] := 7;
   // PSTT[16] := 14;
   // PSTT[17] := 15;
   // PSTT[18] := 3;
   // PSTT[19] := 16;
   // PSTT[20] := 17;
   // PSTT[21] := 18;
   // PSTT[22] := 19;
   // PSTT[23] := 20;
   // PSTT[24] := 21;
   // PSTT[25] := 22;
   // PSTT[26] := 19;
   // PSTT[27] := 23;
   // PSTT[28] := 24;
   // PSTT[29] := 25;
   // PSTT[30] := 19;
   // PSTT[31] := 26;
   // PSTT[32] := 27;
   // PSTT[33] := 3;
   // PSTT[34] := 28;
   // PSTT[35] := 29;
   // NSTT[7] := 8;
   // NSTT[8] := 9;
   // NSTT[9] := 10;
   // NSTT[10] := 3;
   // NSTT[11] := 11;
   // NSTT[12] := 12;
   // NSTT[13] := 13;
   // NSTT[14] := 19;
   // NSTT[15] := 14;
   // NSTT[16] := 15;
   // NSTT[17] := 7;
   // NSTT[18] := 16;
   // NSTT[19] := 17;
   // NSTT[20] := 18;
   // NSTT[21] := 19;
   // NSTT[22] := 20;
   // NSTT[23] := 21;
   // NSTT[24] := 22;
   // NSTT[25] := 7;
   // NSTT[26] := 23;
   // NSTT[27] := 24;
   // NSTT[28] := 25;
   // NSTT[29] := 3;
   // NSTT[30] := 26;
   // NSTT[31] := 27;
   // NSTT[32] := 19;
   // NSTT[33] := 28;
   // NSTT[34] := 29;
   // NSTT[35] := 3;
   // ASSJ[7] := 7;
   // ASSJ[8] := 8;
   // ASSJ[9] := 9;
   // ASSJ[10] := 10;
   // ASSJ[11] := 11;
   // ASSJ[12] := 12;
   // ASSJ[13] := 13;
   // ASSJ[14] := 14;
   // ASSJ[15] := 15;
   // ASSJ[16] := 16;
   // ASSJ[17] := 17;
   // ASSJ[18] := 18;
   // ASSJ[19] := 19;
   // ASSJ[20] := 20;
   // ASSJ[21] := 21;
   // ASSJ[22] := 22;
   // ASSJ[23] := 23;
   // ASSJ[24] := 24;
   // ASSJ[25] := 25;
   // ASSJ[26] := 26;
   // ASSJ[27] := 27;
   // ASSJ[28] := 28;
   // ASSJ[29] := 29;
   // ASSB[7] := 7;
   // ASSB[8] := 8;
   // ASSB[9] := 9;
   // ASSB[10] := 10;
   // ASSB[11] := 11;
   // ASSB[12] := 12;
   // ASSB[13] := 13;
   // ASSB[14] := 14;
   // ASSB[15] := 15;
   // ASSB[16] := 16;
   // ASSB[17] := 17;
   // ASSB[18] := 18;
   // ASSB[19] := 19;
   // ASSB[20] := 20;
   // ASSB[21] := 21;
   // ASSB[22] := 22;
   // ASSB[23] := 23;
   // ASSB[24] := 24;
   // ASSB[25] := 25;
   // ASSB[26] := 26;
   // ASSB[27] := 27;
   // ASSB[28] := 28;
   // ASSB[29] := 29;
   // PTTS[7] := 6;
   // PTTS[8] := 7;
   // PTTS[9] := 8;
   // PTTS[10] := 9;
   // PTTS[11] := 11;
   // PTTS[12] := 12;
   // PTTS[13] := 13;
   // PTTS[14] := 15;
   // PTTS[15] := 16;
   // PTTS[16] := 18;
   // PTTS[17] := 19;
   // PTTS[18] := 20;
   // PTTS[19] := 21;
   // PTTS[20] := 22;
   // PTTS[21] := 23;
   // PTTS[22] := 24;
   // PTTS[23] := 26;
   // PTTS[24] := 27;
   // PTTS[25] := 28;
   // PTTS[26] := 30;
   // PTTS[27] := 31;
   // PTTS[28] := 33;
   // PTTS[29] := 34;
   // NTTS[7] := 7;
   // NTTS[8] := 8;
   // NTTS[9] := 9;
   // NTTS[10] := 10;
   // NTTS[11] := 12;
   // NTTS[12] := 13;
   // NTTS[13] := 14;
   // NTTS[14] := 16;
   // NTTS[15] := 17;
   // NTTS[16] := 19;
   // NTTS[17] := 20;
   // NTTS[18] := 21;
   // NTTS[19] := 22;
   // NTTS[20] := 23;
   // NTTS[21] := 24;
   // NTTS[22] := 25;
   // NTTS[23] := 27;
   // NTTS[24] := 28;
   // NTTS[25] := 29;
   // NTTS[26] := 31;
   // NTTS[27] := 32;
   // NTTS[28] := 34;
   // NTTS[29] := 35;
   // SW_SQTS[8] := 2;
   // SW_SQTS[9] := 2;
   // SW_SQTS[10] := 2;
   // SW_SQTS[11] := 3;
   // SW_SQTS[12] := 3;
   // SW_SQTS[13] := 3;
   // SW_SQTS[14] := 4;
   // SW_SQTS[15] := 4;
   // SW_SQTS[16] := 5;
   // SW_SQTS[17] := 6;
   // SW_SQTS[18] := 6;
   // SW_SQTS[19] := 6;
   // SW_SQTS[20] := 7;
   // SW_SQTS[21] := 7;
   // SW_SQTS[22] := 7;
   // SW_SQTS[23] := 8;
   // SW_SQTS[24] := 9;
   // SW_SQTS[25] := 9;
   // SW_SQTS[26] := 10;
   // SW_SQTS[27] := 10;
   // SW_SQTS[28] := 11;
   // SW_SQTS[29] := 11;
   // SW_SQTS[7] := 1;
   // SW_SQTS[6] := 1;
   // SW_SQTS[5] := 1;
   // SW_SQTS[4] := 1;
   // LSTT[36] := 4;
   // ATAJ[36] := 36;
   // ATAB[36] := 19;
   // PSTT[36] := 16;
   // NSTT[36] := 4;
   // LSTT[37] := 20;
   // ATAJ[37] := 37;
   // ATAB[37] := 27;
   // PSTT[37] := 23;
   // NSTT[37] := 20;
BEGIN
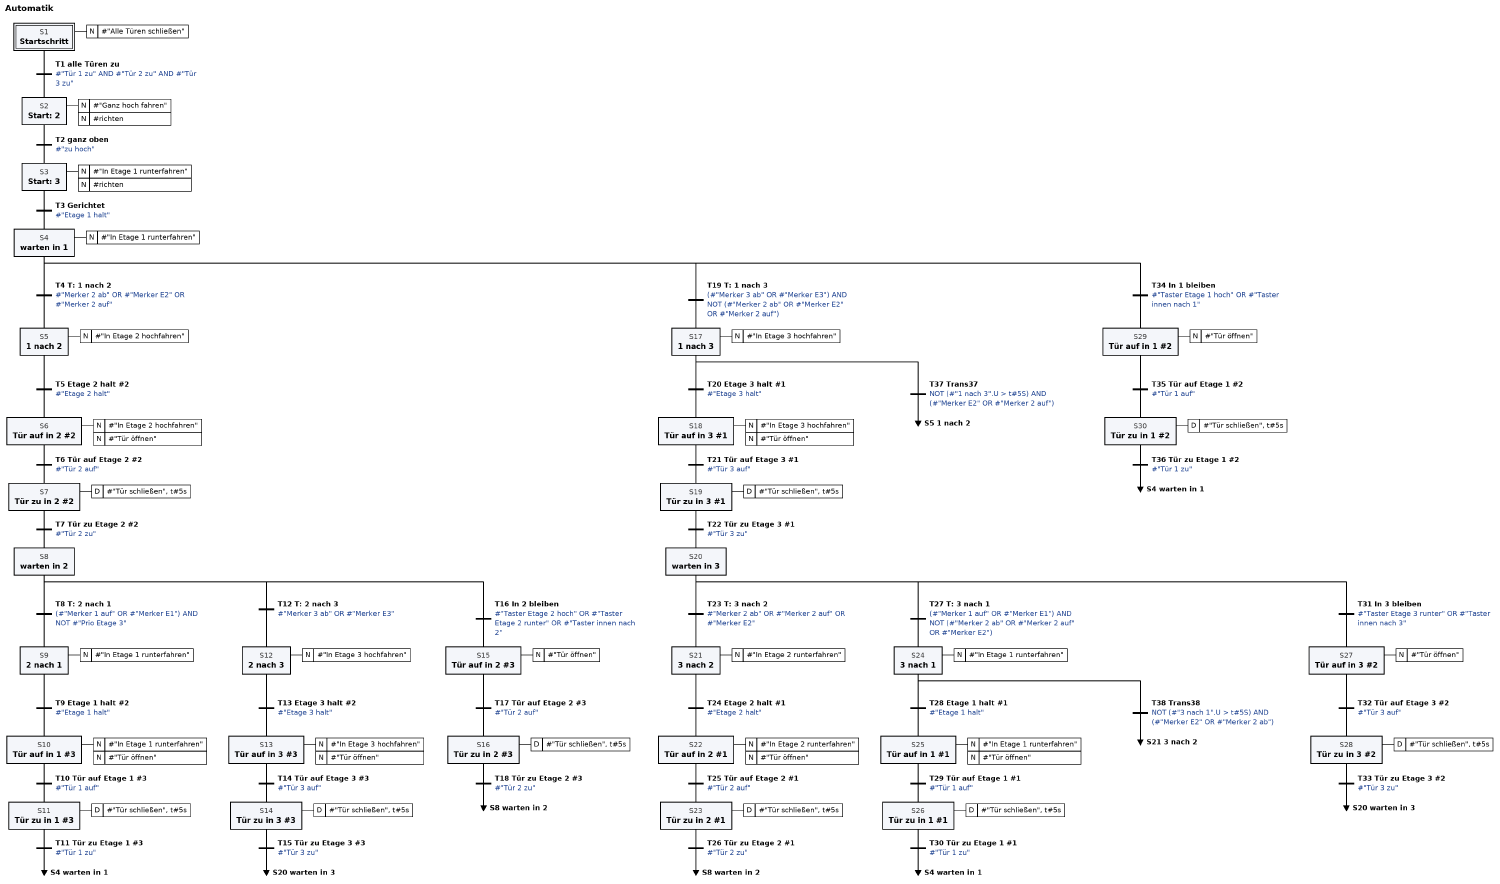
   // sequencer 1
   INITIAL_STEP Startschritt:   // S1, max time T#10S, warning time T#7S
      // Ganz hoch fahren
              N    #"Alle Türen schließen"
   END_STEP
   TRANSITION "alle Türen zu" FROM Startschritt TO "Start: 2"   // T1: alle Türen zu
      := #"Tür 1 zu" AND #"Tür 2 zu" AND #"Tür 3 zu";
   END_TRANSITION
   STEP "Start: 2":   // S2, max time T#10S, warning time T#7S
      // nach Etage 3 fahren
              N    #"Ganz hoch fahren"
              N    #richten
   END_STEP
   TRANSITION "ganz oben" FROM "Start: 2" TO "Start: 3"   // T2: in Etage 3 angekommen
      := #"zu hoch";
   END_TRANSITION
   STEP "Start: 3":   // S3, max time T#10S, warning time T#7S
      // Tür 3 schließen
              N    #"In Etage 1 runterfahren"
              N    #richten
   END_STEP
   TRANSITION Gerichtet FROM "Start: 3" TO "warten in 1"   // T3
      := #"Etage 1 halt";
   END_TRANSITION
   STEP "warten in 1":   // S4, max time T#10S, warning time T#7S
              N    #"In Etage 1 runterfahren"
   END_STEP
   TRANSITION "T: 1 nach 2" FROM "warten in 1" TO "1 nach 2"   // T4
      := #"Merker 2 ab" OR #"Merker E2" OR #"Merker 2 auf";
   END_TRANSITION
   TRANSITION "T: 1 nach 3" FROM "warten in 1" TO "1 nach 3"   // T19
      := (#"Merker 3 ab" OR #"Merker E3") AND NOT (#"Merker 2 ab" OR #"Merker E2" OR #"Merker 2 auf");
   END_TRANSITION
   TRANSITION "In 1 bleiben" FROM "warten in 1" TO "Tür auf in 1 #2"   // T34
      := #"Taster Etage 1 hoch" OR #"Taster innen nach 1";
   END_TRANSITION
   STEP "1 nach 3":   // S17, max time T#10S, warning time T#7S
      // eins nach 3
              N    #"In Etage 3 hochfahren"
   END_STEP
   TRANSITION "Etage 3 halt #1" FROM "1 nach 3" TO "Tür auf in 3 #1"   // T20
      := #"Etage 3 halt";
   END_TRANSITION
   TRANSITION Trans37 FROM "1 nach 3" TO "1 nach 2"   // T37, jump
      := NOT (#"1 nach 3".U > t#5S) AND (#"Merker E2" OR #"Merker 2 auf");
   END_TRANSITION
   STEP "Tür auf in 3 #1":   // S18, max time T#10S, warning time T#7S
              N    #"In Etage 3 hochfahren"
              N    #"Tür öffnen"
   END_STEP
   TRANSITION "Tür auf Etage 3 #1" FROM "Tür auf in 3 #1" TO "Tür zu in 3 #1"   // T21
      := #"Tür 3 auf";
   END_TRANSITION
   STEP "Tür zu in 3 #1":   // S19, max time T#10S, warning time T#7S
              D    #"Tür schließen", t#5s
   END_STEP
   TRANSITION "Tür zu Etage 3 #1" FROM "Tür zu in 3 #1" TO "warten in 3"   // T22
      := #"Tür 3 zu";
   END_TRANSITION
   STEP "1 nach 2":   // S5, max time T#10S, warning time T#7S
              N    #"In Etage 2 hochfahren"
   END_STEP
   TRANSITION "Etage 2 halt #2" FROM "1 nach 2" TO "Tür auf in 2 #2"   // T5
      := #"Etage 2 halt";
   END_TRANSITION
   STEP "Tür auf in 2 #2":   // S6, max time T#10S, warning time T#7S
              N    #"In Etage 2 hochfahren"
              N    #"Tür öffnen"
   END_STEP
   TRANSITION "Tür auf Etage 2 #2" FROM "Tür auf in 2 #2" TO "Tür zu in 2 #2"   // T6
      := #"Tür 2 auf";
   END_TRANSITION
   STEP "Tür zu in 2 #2":   // S7, max time T#10S, warning time T#7S
              D    #"Tür schließen", t#5s
   END_STEP
   TRANSITION "Tür zu Etage 2 #2" FROM "Tür zu in 2 #2" TO "warten in 2"   // T7
      := #"Tür 2 zu";
   END_TRANSITION
   STEP "warten in 3":   // S20, max time T#10S, warning time T#7S
   END_STEP
   TRANSITION "T: 3 nach 2" FROM "warten in 3" TO "3 nach 2"   // T23
      := #"Merker 2 ab" OR #"Merker 2 auf" OR #"Merker E2";
   END_TRANSITION
   TRANSITION "T: 3 nach 1" FROM "warten in 3" TO "3 nach 1"   // T27
      := (#"Merker 1 auf" OR #"Merker E1") AND NOT (#"Merker 2 ab" OR #"Merker 2 auf" OR #"Merker E2");
   END_TRANSITION
   TRANSITION "In 3 bleiben" FROM "warten in 3" TO "Tür auf in 3 #2"   // T31
      := #"Taster Etage 3 runter" OR #"Taster innen nach 3";
   END_TRANSITION
   STEP "warten in 2":   // S8, max time T#10S, warning time T#7S
   END_STEP
   TRANSITION "T: 2 nach 1" FROM "warten in 2" TO "2 nach 1"   // T8
      := (#"Merker 1 auf" OR #"Merker E1") AND NOT #"Prio Etage 3";
   END_TRANSITION
   TRANSITION "T: 2 nach 3" FROM "warten in 2" TO "2 nach 3"   // T12
      := #"Merker 3 ab" OR #"Merker E3";
   END_TRANSITION
   TRANSITION "In 2 bleiben" FROM "warten in 2" TO "Tür auf in 2 #3"   // T16
      := #"Taster Etage 2 hoch" OR #"Taster Etage 2 runter" OR #"Taster innen nach 2";
   END_TRANSITION
   STEP "Tür auf in 1 #2":   // S29, max time T#10S, warning time T#7S
              N    #"Tür öffnen"
   END_STEP
   TRANSITION "Tür auf Etage 1 #2" FROM "Tür auf in 1 #2" TO "Tür zu in 1 #2"   // T35
      := #"Tür 1 auf";
   END_TRANSITION
   STEP "Tür zu in 1 #2":   // S30, max time T#10S, warning time T#7S
              D    #"Tür schließen", t#5s
   END_STEP
   TRANSITION "Tür zu Etage 1 #2" FROM "Tür zu in 1 #2" TO "warten in 1"   // T36, jump
      := #"Tür 1 zu";
   END_TRANSITION
   STEP "3 nach 2":   // S21, max time T#10S, warning time T#7S
              N    #"In Etage 2 runterfahren"
   END_STEP
   TRANSITION "Etage 2 halt #1" FROM "3 nach 2" TO "Tür auf in 2 #1"   // T24
      := #"Etage 2 halt";
   END_TRANSITION
   STEP "Tür auf in 2 #1":   // S22, max time T#10S, warning time T#7S
      // Tür auf in 2 #1
              N    #"In Etage 2 runterfahren"
              N    #"Tür öffnen"
   END_STEP
   TRANSITION "Tür auf Etage 2 #1" FROM "Tür auf in 2 #1" TO "Tür zu in 2 #1"   // T25
      := #"Tür 2 auf";
   END_TRANSITION
   STEP "Tür zu in 2 #1":   // S23, max time T#10S, warning time T#7S
              D    #"Tür schließen", t#5s
   END_STEP
   TRANSITION "Tür zu Etage 2 #1" FROM "Tür zu in 2 #1" TO "warten in 2"   // T26, jump
      := #"Tür 2 zu";
   END_TRANSITION
   STEP "3 nach 1":   // S24, max time T#10S, warning time T#7S
              N    #"In Etage 1 runterfahren"
   END_STEP
   TRANSITION "Etage 1 halt #1" FROM "3 nach 1" TO "Tür auf in 1 #1"   // T28
      := #"Etage 1 halt";
   END_TRANSITION
   TRANSITION Trans38 FROM "3 nach 1" TO "3 nach 2"   // T38, jump
      := NOT (#"3 nach 1".U > t#5S) AND (#"Merker E2" OR #"Merker 2 ab");
   END_TRANSITION
   STEP "Tür auf in 1 #1":   // S25, max time T#10S, warning time T#7S
              N    #"In Etage 1 runterfahren"
              N    #"Tür öffnen"
   END_STEP
   TRANSITION "Tür auf Etage 1 #1" FROM "Tür auf in 1 #1" TO "Tür zu in 1 #1"   // T29
      := #"Tür 1 auf";
   END_TRANSITION
   STEP "Tür zu in 1 #1":   // S26, max time T#10S, warning time T#7S
              D    #"Tür schließen", t#5s
   END_STEP
   TRANSITION "Tür zu Etage 1 #1" FROM "Tür zu in 1 #1" TO "warten in 1"   // T30, jump
      := #"Tür 1 zu";
   END_TRANSITION
   STEP "Tür auf in 3 #2":   // S27, max time T#10S, warning time T#7S
              N    #"Tür öffnen"
   END_STEP
   TRANSITION "Tür auf Etage 3 #2" FROM "Tür auf in 3 #2" TO "Tür zu in 3 #2"   // T32
      := #"Tür 3 auf";
   END_TRANSITION
   STEP "Tür zu in 3 #2":   // S28, max time T#10S, warning time T#7S
              D    #"Tür schließen", t#5s
   END_STEP
   TRANSITION "Tür zu Etage 3 #2" FROM "Tür zu in 3 #2" TO "warten in 3"   // T33, jump
      := #"Tür 3 zu";
   END_TRANSITION
   STEP "2 nach 1":   // S9, max time T#10S, warning time T#7S
              N    #"In Etage 1 runterfahren"
   END_STEP
   TRANSITION "Etage 1 halt #2" FROM "2 nach 1" TO "Tür auf in 1 #3"   // T9
      := #"Etage 1 halt";
   END_TRANSITION
   STEP "2 nach 3":   // S12, max time T#10S, warning time T#7S
              N    #"In Etage 3 hochfahren"
   END_STEP
   TRANSITION "Etage 3 halt #2" FROM "2 nach 3" TO "Tür auf in 3 #3"   // T13
      := #"Etage 3 halt";
   END_TRANSITION
   STEP "Tür auf in 2 #3":   // S15, max time T#10S, warning time T#7S
              N    #"Tür öffnen"
   END_STEP
   TRANSITION "Tür auf Etage 2 #3" FROM "Tür auf in 2 #3" TO "Tür zu in 2 #3"   // T17
      := #"Tür 2 auf";
   END_TRANSITION
   STEP "Tür zu in 2 #3":   // S16, max time T#10S, warning time T#7S
              D    #"Tür schließen", t#5s
   END_STEP
   TRANSITION "Tür zu Etage 2 #3" FROM "Tür zu in 2 #3" TO "warten in 2"   // T18, jump
      := #"Tür 2 zu";
   END_TRANSITION
   STEP "Tür auf in 1 #3":   // S10, max time T#10S, warning time T#7S
              N    #"In Etage 1 runterfahren"
              N    #"Tür öffnen"
   END_STEP
   TRANSITION "Tür auf Etage 1 #3" FROM "Tür auf in 1 #3" TO "Tür zu in 1 #3"   // T10
      := #"Tür 1 auf";
   END_TRANSITION
   STEP "Tür zu in 1 #3":   // S11, max time T#10S, warning time T#7S
              D    #"Tür schließen", t#5s
   END_STEP
   TRANSITION "Tür zu Etage 1 #3" FROM "Tür zu in 1 #3" TO "warten in 1"   // T11, jump
      := #"Tür 1 zu";
   END_TRANSITION
   STEP "Tür auf in 3 #3":   // S13, max time T#10S, warning time T#7S
              N    #"In Etage 3 hochfahren"
              N    #"Tür öffnen"
   END_STEP
   TRANSITION "Tür auf Etage 3 #3" FROM "Tür auf in 3 #3" TO "Tür zu in 3 #3"   // T14
      := #"Tür 3 auf";
   END_TRANSITION
   STEP "Tür zu in 3 #3":   // S14, max time T#10S, warning time T#7S
              D    #"Tür schließen", t#5s
   END_STEP
   TRANSITION "Tür zu Etage 3 #3" FROM "Tür zu in 3 #3" TO "warten in 3"   // T15, jump
      := #"Tür 3 zu";
   END_TRANSITION
END_FUNCTION_BLOCK

FUNCTION_BLOCK "7-Segment Anzeige"   // FB7, SCL
{ S7_Optimized_Access := 'TRUE' }
VERSION : 0.1
   VAR_INPUT
      "Etage 1 halt" : Bool;   // Endlage Etage 1
      "Etage 2 halt" : Bool;   // Endlage Etage 2
      "Etage 3 halt" : Bool;   // Endlage Etage 3
   END_VAR
   VAR_OUTPUT
      "7S A" : Bool;   // Segment a
      "7S B" : Bool;   // Segment b
      "7S C" : Bool;   // Segment c
      "7S D" : Bool;   // Segment d
      "7S E" : Bool;   // Segment e
      "7S F" : Bool;   // Segment f
      "7S G" : Bool;   // Segment g
   END_VAR
   VAR
      Etage : Int;   // Etagennummer
   END_VAR
BEGIN
   (*Umwandlung Etagennummer in Int*)
   IF #"Etage 1 halt" THEN
       #Etage := 1;
   ELSIF #"Etage 2 halt" THEN
       #Etage := 2;
   ELSIF #"Etage 3 halt" THEN
       #Etage := 3;
   END_IF;

   (*Anzeige Etagennummer*)
   IF #"Etage 1 halt" THEN
       #"7S A" := 0;
       #"7S B" := 1;
       #"7S C" := 1;
       #"7S D" := 0;
       #"7S E" := 0;
       #"7S F" := 0;
       #"7S G" := 0;
   END_IF;

   IF #"Etage 2 halt" THEN
       #"7S A" := 1;
       #"7S B" := 1;
       #"7S C" := 0;
       #"7S D" := 1;
       #"7S E" := 1;
       #"7S F" := 0;
       #"7S G" := 1;
   END_IF;

   IF #"Etage 3 halt" THEN
       #"7S A" := 1;
       #"7S B" := 1;
       #"7S C" := 1;
       #"7S D" := 1;
       #"7S E" := 0;
       #"7S F" := 0;
       #"7S G" := 1;
   END_IF;
END_FUNCTION_BLOCK

FUNCTION_BLOCK "LED-Funktionen"   // FB8, SCL
{ S7_Optimized_Access := 'TRUE' }
VERSION : 0.1
   VAR_INPUT
      "Merker Etage 1" : Bool;   // Anforderung Etage 1 innen
      "Merker Etage 2" : Bool;   // Anforderung Etage 2 innen
      "Merker Etage 3" : Bool;   // Anforderung Etage 3 innen
      "Merker Etage 1 Auf" : Bool;   // Anforderung Etage 1 hoch
      "Merker Etage 2 Auf" : Bool;   // Anforderung Etage 2 hoch
      "Merker Etage 2 Ab" : Bool;   // Anforderung Etage 2 runter
      "Merker Etage 3 Ab" : Bool;   // Anforderung Etage 3 runter
   END_VAR
   VAR_OUTPUT
      "LED Etage 1" : Bool;   // LED Kabine Etage 1
      "LED Etage 2" : Bool;   // LED Kabine Etage 2
      "LED Etage 3" : Bool;   // LED Kabine Etage 3
      "LED Etage 1 Auf" : Bool;   // LED Etage 1 hoch
      "LED Etage 2 Auf" : Bool;   // LED Etage 2 hoch
      "LED Etage 2 Ab" : Bool;   // LED Etage 2 runter
      "LED Etage 3 Ab" : Bool;   // LED Etage 3 runter
   END_VAR
   VAR
      "Blinken aktiv" : Bool;   // LEDs blinken
   END_VAR
BEGIN
   (*Funktion blinken*)
   #"Blinken aktiv" :=  ("Automatik_DB".Startschritt.X OR "Automatik_DB"."Start: 2".X OR "Automatik_DB"."Start: 3".X OR "Handbetrieb_DB"."Hand aktiv") AND "Clock_1Hz";

   (*Ansteuerung LEDs*)
   #"LED Etage 1" := #"Merker Etage 1" AND NOT #"Blinken aktiv" OR #"Blinken aktiv";
   #"LED Etage 2" := #"Merker Etage 2" AND NOT #"Blinken aktiv" OR #"Blinken aktiv";
   #"LED Etage 3" := #"Merker Etage 3" AND NOT #"Blinken aktiv" OR #"Blinken aktiv";
   #"LED Etage 1 Auf" := #"Merker Etage 1 Auf" AND NOT #"Blinken aktiv" OR #"Blinken aktiv";
   #"LED Etage 2 Auf" := #"Merker Etage 2 Auf" AND NOT #"Blinken aktiv" OR #"Blinken aktiv";
   #"LED Etage 2 Ab" := #"Merker Etage 2 Ab" AND NOT #"Blinken aktiv" OR #"Blinken aktiv";
   #"LED Etage 3 Ab" := #"Merker Etage 3 Ab" AND NOT #"Blinken aktiv" OR #"Blinken aktiv";
END_FUNCTION_BLOCK

FUNCTION_BLOCK "Merker"   // FB9, SCL
{ S7_Optimized_Access := 'TRUE' }
VERSION : 0.1
   VAR_INPUT
      "Taster Etage I (innen)" : Bool;   // Taster Etage 1 innen
      "Taster Etage II (innen)" : Bool;   // Taster Etage 2 innen
      "Taster Etage III (innen)" : Bool;   // Taster Etage 3 innen
      "Taster Etage I Auf" : Bool;   // Taster Etage 1 hoch
      "Taster Etage II Auf" : Bool;   // Taster Etage 2 hoch
      "Taster Etage II Ab" : Bool;   // Taster Etage 2 runter
      "Taster Etage III Ab" : Bool;   // Taster Etage 3 runter
      "Etage 1 halt" : Bool;   // Etage 1 halt
      "Etage 2 halt" : Bool;   // Etage 2 halt
      "Etage 3 halt" : Bool;   // Etage 3 halt
      Automatikbetrieb : Bool;   // Automatikbetrieb
      "Not-Aus" : Bool;   // Notaus
   END_VAR
   VAR_OUTPUT
      "Merker Etage 1" : Bool;   // Anforderung Etage 1 innen
      "Merker Etage 2" : Bool;   // Anforderung Etage 2 innen
      "Merker Etage 3" : Bool;   // Anforderung Etage 3 innen
      "Merker Etage 1 Auf" : Bool;   // Anforderung Etage 1 hoch
      "Merker Etage 2 Auf" : Bool;   // Anforderung Etage 2 hoch
      "Merker Etage 2 Ab" : Bool;   // Anforderung Etage 2 runter
      "Merker Etage 3 Ab" : Bool;   // Anforderung Etage 3 runter
   END_VAR
   VAR
      Tür1 : String;   // OPC-UA Text Tür 1
      Tür2 : String;   // OPC-UA Text Tür 2
      Tür3 : String;   // OPC-UA Text Tür 3
      Betriebsart : String;   // OPC-UA Text Betriebsart
      Fahrt_Fahrstuhl : String;   // OPC-UA Text Fahrt Fahrstuhl
   END_VAR
BEGIN
   (*Anforderung Kabine Etage 1*)
   IF #"Taster Etage I (innen)" THEN
       #"Merker Etage 1":=1;
   END_IF;
   IF #"Etage 1 halt" OR #"Not-Aus" OR #Automatikbetrieb = 0 THEN
       #"Merker Etage 1":=0;
   END_IF;

   (*Anforderung Kabine Etage 2*)
   IF #"Taster Etage II (innen)" THEN
       #"Merker Etage 2" := 1;
   END_IF;
   IF (#"Etage 2 halt" OR #"Not-Aus") AND "Automatik_DB"."1 nach 3".X=0 AND "Automatik_DB"."3 nach 1".X=0 OR #Automatikbetrieb = 0 THEN
       #"Merker Etage 2" := 0;
   END_IF;

   (*Anforderung Kabine Etage 3*)
   IF #"Taster Etage III (innen)" THEN
       #"Merker Etage 3" := 1;
   END_IF;
   IF #"Etage 3 halt" OR #"Not-Aus" OR #Automatikbetrieb = 0 THEN
       #"Merker Etage 3" := 0;
   END_IF;

   (*Anforderung Etage 1 hoch*)
   IF #"Taster Etage I Auf" THEN
       #"Merker Etage 1 Auf" := 1;
   END_IF;
   IF #"Etage 1 halt" OR #"Not-Aus" OR #Automatikbetrieb = 0 THEN
       #"Merker Etage 1 Auf" := 0;
   END_IF;

   (*Anforderung Etage 2 hoch*)
   IF #"Taster Etage II Auf" THEN
       #"Merker Etage 2 Auf" := 1;
   END_IF;
   IF (#"Etage 2 halt" OR #"Not-Aus") AND "Automatik_DB"."1 nach 3".X=0 AND "Automatik_DB"."3 nach 1".X=0 OR #Automatikbetrieb = 0 THEN
       #"Merker Etage 2 Auf" := 0;
   END_IF;

   (*Anforderung Etage 2 runter*)
   IF #"Taster Etage II Ab" THEN
       #"Merker Etage 2 Ab" := 1;
   END_IF;
   IF (#"Etage 2 halt" OR #"Not-Aus") AND "Automatik_DB"."1 nach 3".X=0 AND "Automatik_DB"."3 nach 1".X=0 OR #Automatikbetrieb = 0 THEN
       #"Merker Etage 2 Ab" := 0;
   END_IF;

   (*Anforderung Etage 3 runter*)
   IF #"Taster Etage III Ab" THEN
       #"Merker Etage 3 Ab" := 1;
   END_IF;
   IF #"Etage 3 halt" OR #"Not-Aus" OR #Automatikbetrieb = 0 THEN
       #"Merker Etage 3 Ab" := 0;
   END_IF;


   (*Statics für OPC-UA*)
   IF "Endlage Tür I Auf" THEN
       #Tür1 := 'offen';
   ELSIF "Endlage Tür I Zu" THEN
       #Tür1 := 'geschlossen';
   END_IF;
   IF "Endlage Tür II Auf" THEN
       #Tür2 := 'offen';
   ELSIF "Endlage Tür II Zu" THEN
       #Tür2 := 'geschlossen';
   END_IF;
   IF "Endlage Tür III Auf" THEN
       #Tür3 := 'offen';
   ELSIF "Endlage Tür III Zu" THEN
       #Tür3 := 'geschlossen';
   END_IF;
   IF ("Automatikbetrieb" AND "Not-Aus" AND NOT "Automatik_DB".richten) THEN
       #Betriebsart := 'Automatikbetrieb';
   ELSIF NOT "Not-Aus" THEN
       #Betriebsart := 'Notaus';
   ELSIF ("Automatik_DB".richten AND "Not-Aus") THEN
       #Betriebsart := 'Richtbetrieb';
   ELSE
       #Betriebsart := 'Handbetrieb';
   END_IF;
   IF "Hubmotor langsam Heben" THEN
       #Fahrt_Fahrstuhl := 'langsam hoch';
   ELSIF "Hubmotor schnell Heben" THEN
       #Fahrt_Fahrstuhl := 'schnell hoch';
   ELSIF "Hubmotor schnell Senken" THEN
       #Fahrt_Fahrstuhl := 'schnell runter';
   ELSIF "Hubmotor schnell Senken" THEN
       #Fahrt_Fahrstuhl := 'schnell runter';
   ELSE
       #Fahrt_Fahrstuhl := 'nicht';
   END_IF;
END_FUNCTION_BLOCK

FUNCTION_BLOCK "Zeitbaustein Priorisierung"   // FB10, FBD
TITLE = Zeitbaustein Priorisierung
{ S7_Optimized_Access := 'TRUE' }
VERSION : 0.1
// Priorisierung der zuerst gewählten Etage, wenn in Etage 2 im Automatikbetrieb
   VAR_INPUT
      "Endlage Etage I Halt" : Bool;   // Endlage Etage 1
      "Endlage Etage II Halt" : Bool;   // Endlage Etage 2
      "Endlage Etage III Halt" : Bool;   // Endlage Etage 3
      "Not-Aus" : Bool;   // Notaus
      "Merker Etage I" : Bool;   // Anforderung Etage 1 innen
      "Merker Etage II" : Bool;   // Anforderung Etage 2 innen
      "Merker Etage III" : Bool;   // Anforderung Etage 3 innen
      "Merker Etage I Auf" : Bool;   // Anforderung Etage 1 hoch
      "Merker Etage II Auf" : Bool;   // Anforderung Etage 2 hoch
      "Merker Etage II Ab" : Bool;   // Anforderung Etage 2 runter
      "Merker Etage III Ab" : Bool;   // Anforderung Etage 3 runter
   END_VAR
   VAR_OUTPUT
      "Prio 3" : Bool;   // Priorisierung Etage 3
   END_VAR
BEGIN

REGION Network 1: Timer Anforderung Etage 1
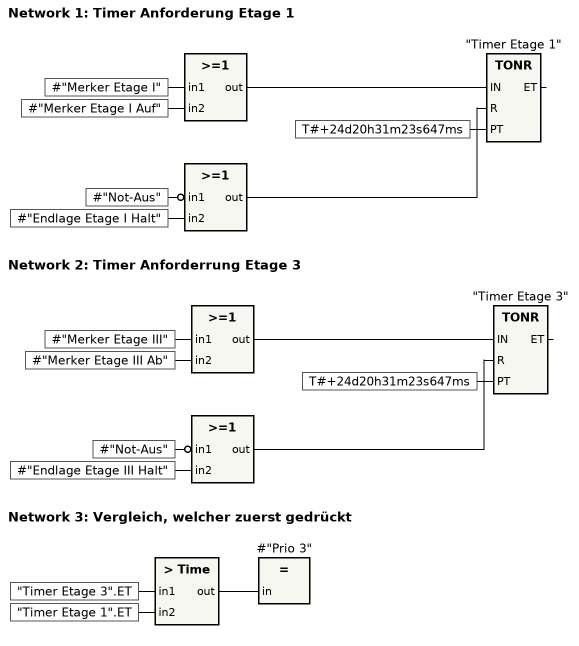
   "Timer Etage 1".TONR(IN := #"Merker Etage I" OR #"Merker Etage I Auf",
                        R := NOT #"Not-Aus" OR #"Endlage Etage I Halt",
                        PT := T#+24d20h31m23s647ms);
END_REGION

REGION Network 2: Timer Anforderrung Etage 3
   "Timer Etage 3".TONR(IN := #"Merker Etage III" OR #"Merker Etage III Ab",
                        R := NOT #"Not-Aus" OR #"Endlage Etage III Halt",
                        PT := T#+24d20h31m23s647ms);
END_REGION

REGION Network 3: Vergleich, welcher zuerst gedrückt
   #"Prio 3" := "Timer Etage 3".ET > "Timer Etage 1".ET;
END_REGION
END_FUNCTION_BLOCK

FUNCTION_BLOCK "Handbetrieb"   // FB11, FBD
TITLE = Handbetrieb
{ S7_Optimized_Access := 'TRUE' }
VERSION : 0.1
// Richtet, wenn in keiner bestimmten Endlage
   VAR_INPUT
      "Etage 1 halt" : Bool;   // Etage 1 halt
      "Etage 2 halt" : Bool;   // Etage 2 halt
      "Etage 3 halt" : Bool;   // Etage 3 halt
      "Tür Etage 1 zu" : Bool;   // Endlage Tür Etage 1 zu
      "Tür Etage 2 zu" : Bool;   // Endlage Tür Etage 2 zu
      "Tür Etage 3 zu" : Bool;   // Endlage Tür Etage 3 zu
      "Tür Etage 1 auf" : Bool;   // Endlage Tür Etage 1 auf
      "Tür Etage 2 auf" : Bool;   // Endlage Tür Etage 2 auf
      "Tür Etage 3 auf" : Bool;   // Endlage Tür Etage 3 auf
      "Taster Hand hoch" : Bool;   // Taster Hand hoch
      "Taster Hand runter" : Bool;   // Taster Hand runter
      "Taster Hand auf" : Bool;   // Taster Hand auf
      "Taster Hand zu" : Bool;   // Taster Hand zu
      "Not-Aus" : Bool;   // Notaus
      "zu hoch" : Bool;   // Fahrstuhl zu hoch
      "Automatikbetrieb Schalter" : Bool;   // Schalter Automatik
   END_VAR
   VAR_OUTPUT
      "In Etage 1 runterfahren" : Bool;   // In Etage 1 runterfahren
      "In Etage 2 runterfahren" : Bool;   // In Etage 2 runterfahren
      "In Etage 2 hochfahren" : Bool;   // In Etage 2 hochfahren
      "In Etage 3 hochfahren" : Bool;   // In Etage 3 hochfahren
      "Tür zu" : Bool;   // Tür zu
      "Tür auf" : Bool;   // Tür auf
   END_VAR
   VAR
      M1 : Bool;   // Merker 1
      M2 : Bool;   // Merker 2
      M3 : Bool;   // Merker 3
      M4 : Bool;   // Merker 4
      M5 : Bool;   // Merker 5
      M6 : Bool;   // Merker 6
      "Hand aktiv" : Bool;   // Hand aktiv
      "Alle Türen zu" : Bool;   // Alle Türen zu
      "Kein Motor fährt" : Bool;   // Kein Motor fährt
      "Automatik neg. Flanke" : Bool;   // Automatik neg. Flanke
      M7 : Bool;   // Merker 7
      "Handbetrieb neg. Flanke" : Bool;   // Handbetrieb neg. Flanke
      M8 : Bool;   // Merker 8
      "in keiner Endlage" : Bool;   // in keiner Endlage
      "ganz hoch fahren" : Bool;   // ganz hoch fahren
      "in Ausgangspos. fahren" : Bool;   // in Ausgangspos. fahren
      "Kein Richten aktiv" : Bool;   // Kein Richten aktiv
      "Hand Richten beendet Timer" : TON_TIME;   // Timer richten beendet Hand
      "Timer 1" : TON_TIME;   // Timer Etage 1 runter
      "Timer 2" : TON_TIME;   // Timer Etage 3 hoch
      "Timer 3" : TON_TIME;   // Timer Etage 2 runter
      "Timer 4" : TON_TIME;   // Timer Etage 2 hoch
      "Übergabe alle Türen schließen" : Bool;   // alle Türen zu
      "Hand aktiv positive Flanke" : Bool;   // pos Flanke Hand aktiv
   END_VAR
   VAR_TEMP   // added for the SCL form of the ladder/FBD networks
      _w1 : Bool;
   END_VAR
BEGIN

REGION Network 1: Hand aktiv
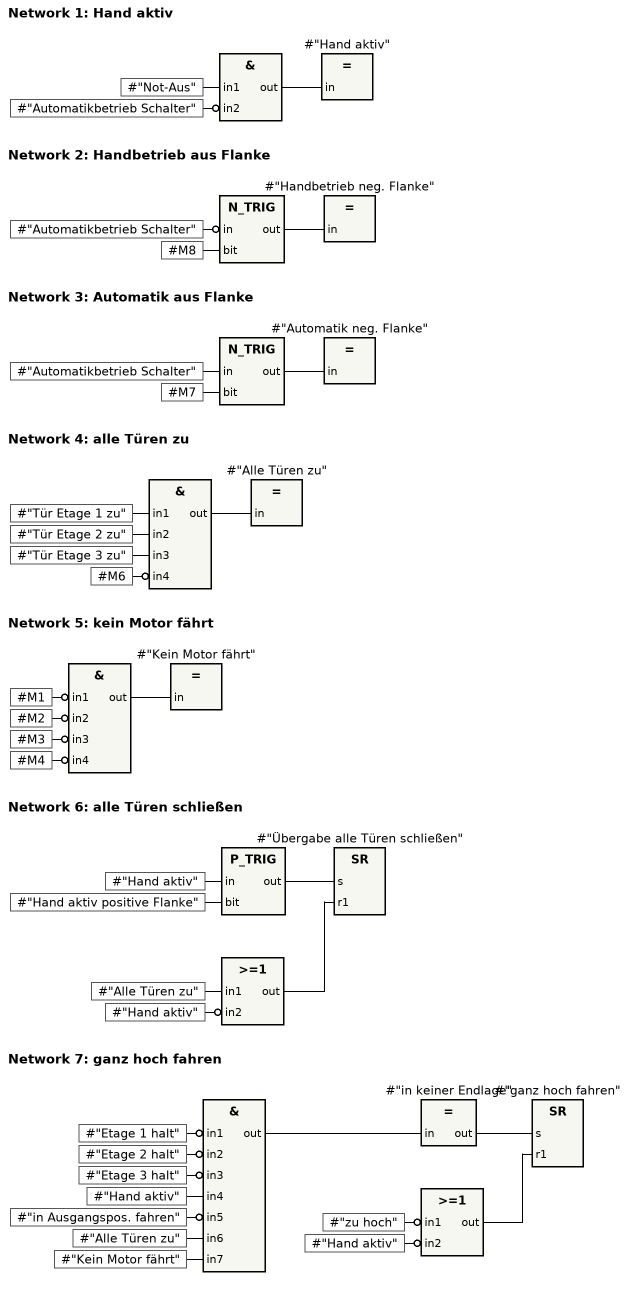
   #"Hand aktiv" := #"Not-Aus" AND NOT #"Automatikbetrieb Schalter";
END_REGION

REGION Network 2: Handbetrieb aus Flanke
   #_w1 := NOT (NOT #"Automatikbetrieb Schalter") AND #M8;   // falling edge
   #M8 := NOT #"Automatikbetrieb Schalter";
   #"Handbetrieb neg. Flanke" := #_w1;
END_REGION

REGION Network 3: Automatik aus Flanke
   #_w1 := NOT #"Automatikbetrieb Schalter" AND #M7;   // falling edge
   #M7 := #"Automatikbetrieb Schalter";
   #"Automatik neg. Flanke" := #_w1;
END_REGION

REGION Network 4: alle Türen zu
   #"Alle Türen zu" := #"Tür Etage 1 zu" AND #"Tür Etage 2 zu" AND #"Tür Etage 3 zu" AND NOT #M6;
END_REGION

REGION Network 5: kein Motor fährt
   #"Kein Motor fährt" := NOT #M1 AND NOT #M2 AND NOT #M3 AND NOT #M4;
END_REGION

REGION Network 6: alle Türen schließen
   #_w1 := #"Hand aktiv" AND NOT #"Hand aktiv positive Flanke";   // rising edge
   #"Hand aktiv positive Flanke" := #"Hand aktiv";
   IF #_w1 THEN
       #"Übergabe alle Türen schließen" := TRUE;   // SR flip-flop
   END_IF;
   IF #"Alle Türen zu" OR NOT #"Hand aktiv" THEN #"Übergabe alle Türen schließen" := FALSE; END_IF;
END_REGION

REGION Network 7: ganz hoch fahren
   #"in keiner Endlage" := NOT #"Etage 1 halt" AND NOT #"Etage 2 halt" AND NOT #"Etage 3 halt" AND #"Hand aktiv" AND NOT #"in Ausgangspos. fahren" AND #"Alle Türen zu" AND #"Kein Motor fährt";
   IF #"in keiner Endlage" THEN
       #"ganz hoch fahren" := TRUE;   // SR flip-flop
   END_IF;
   IF NOT #"zu hoch" OR NOT #"Hand aktiv" THEN #"ganz hoch fahren" := FALSE; END_IF;
END_REGION

REGION Network 8: in Ausgangsposition fahren
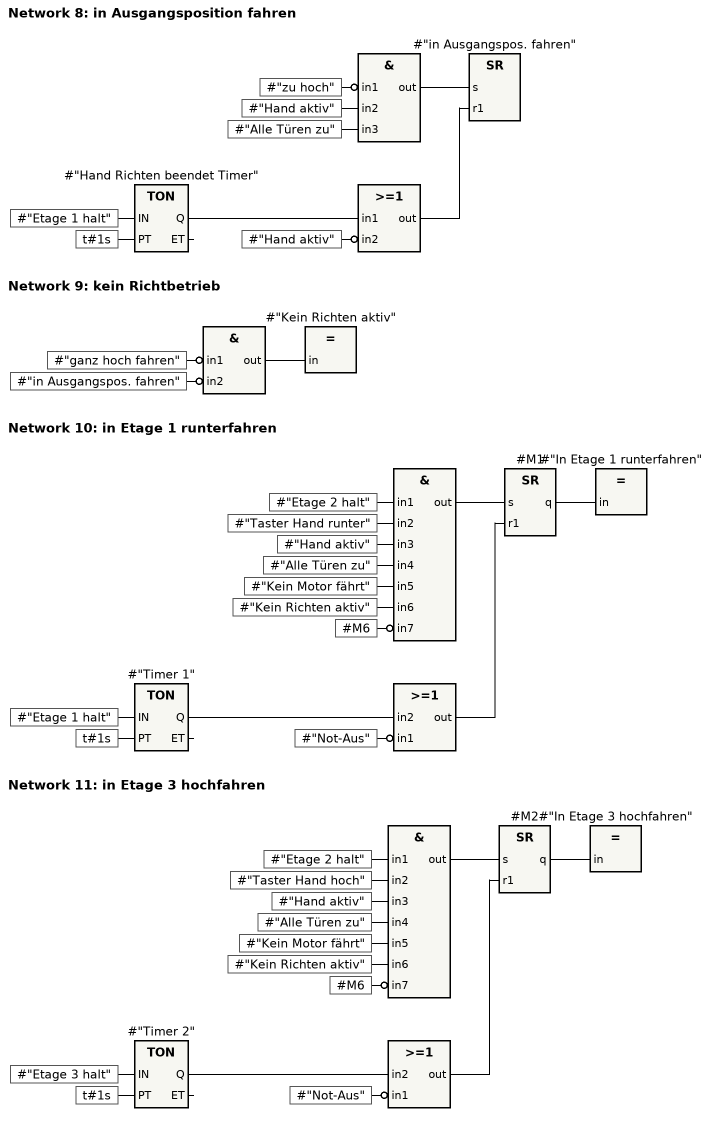
   #"Hand Richten beendet Timer"(IN := #"Etage 1 halt", PT := t#1s);   // TON
   IF NOT #"zu hoch" AND #"Hand aktiv" AND #"Alle Türen zu" THEN
       #"in Ausgangspos. fahren" := TRUE;   // SR flip-flop
   END_IF;
   IF #"Hand Richten beendet Timer".Q OR NOT #"Hand aktiv" THEN #"in Ausgangspos. fahren" := FALSE; END_IF;
END_REGION

REGION Network 9: kein Richtbetrieb
   #"Kein Richten aktiv" := NOT #"ganz hoch fahren" AND NOT #"in Ausgangspos. fahren";
END_REGION

REGION Network 10: in Etage 1 runterfahren
   #"Timer 1"(IN := #"Etage 1 halt", PT := t#1s);   // TON
   IF #"Etage 2 halt" AND #"Taster Hand runter" AND #"Hand aktiv" AND #"Alle Türen zu" AND #"Kein Motor fährt" AND #"Kein Richten aktiv" AND NOT #M6 THEN
       #M1 := TRUE;   // SR flip-flop
   END_IF;
   IF #"Timer 1".Q OR NOT #"Not-Aus" THEN #M1 := FALSE; END_IF;
   #"In Etage 1 runterfahren" := #M1;
END_REGION

REGION Network 11: in Etage 3 hochfahren
   #"Timer 2"(IN := #"Etage 3 halt", PT := t#1s);   // TON
   IF #"Etage 2 halt" AND #"Taster Hand hoch" AND #"Hand aktiv" AND #"Alle Türen zu" AND #"Kein Motor fährt" AND #"Kein Richten aktiv" AND NOT #M6 THEN
       #M2 := TRUE;   // SR flip-flop
   END_IF;
   IF #"Timer 2".Q OR NOT #"Not-Aus" THEN #M2 := FALSE; END_IF;
   #"In Etage 3 hochfahren" := #M2;
END_REGION

REGION Network 12: in Etage 2 runterfahren
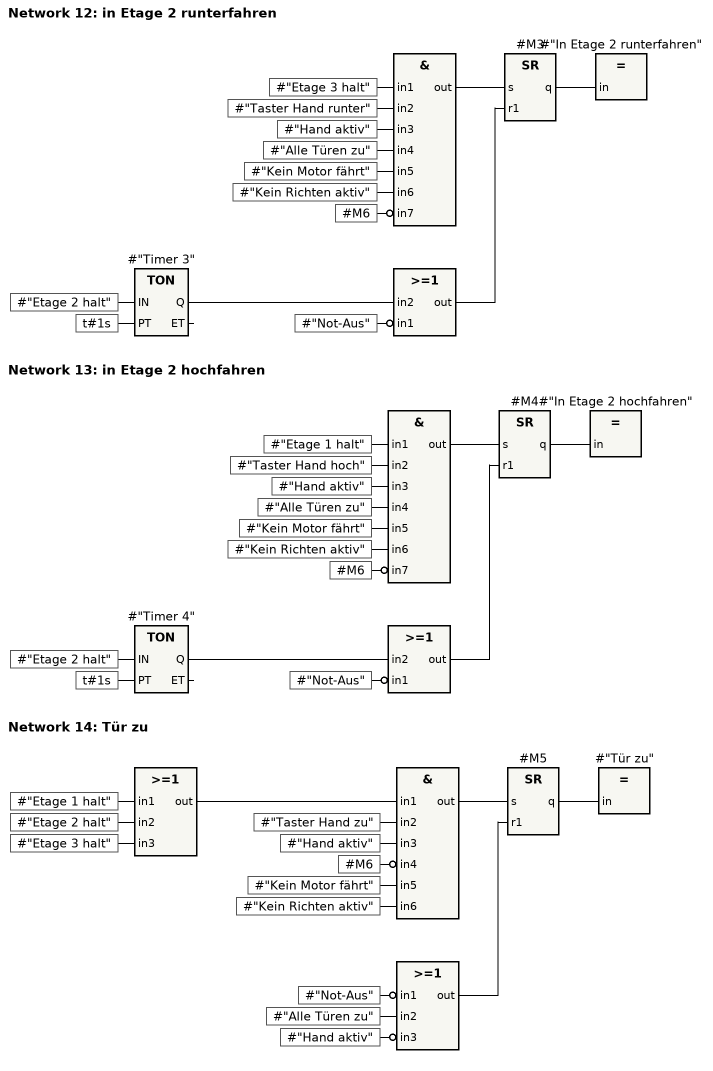
   #"Timer 3"(IN := #"Etage 2 halt", PT := t#1s);   // TON
   IF #"Etage 3 halt" AND #"Taster Hand runter" AND #"Hand aktiv" AND #"Alle Türen zu" AND #"Kein Motor fährt" AND #"Kein Richten aktiv" AND NOT #M6 THEN
       #M3 := TRUE;   // SR flip-flop
   END_IF;
   IF #"Timer 3".Q OR NOT #"Not-Aus" THEN #M3 := FALSE; END_IF;
   #"In Etage 2 runterfahren" := #M3;
END_REGION

REGION Network 13: in Etage 2 hochfahren
   #"Timer 4"(IN := #"Etage 2 halt", PT := t#1s);   // TON
   IF #"Etage 1 halt" AND #"Taster Hand hoch" AND #"Hand aktiv" AND #"Alle Türen zu" AND #"Kein Motor fährt" AND #"Kein Richten aktiv" AND NOT #M6 THEN
       #M4 := TRUE;   // SR flip-flop
   END_IF;
   IF #"Timer 4".Q OR NOT #"Not-Aus" THEN #M4 := FALSE; END_IF;
   #"In Etage 2 hochfahren" := #M4;
END_REGION

REGION Network 14: Tür zu
   IF (#"Etage 1 halt" OR #"Etage 2 halt" OR #"Etage 3 halt") AND #"Taster Hand zu" AND #"Hand aktiv" AND NOT #M6 AND #"Kein Motor fährt" AND #"Kein Richten aktiv" THEN
       #M5 := TRUE;   // SR flip-flop
   END_IF;
   IF NOT #"Not-Aus" OR #"Alle Türen zu" OR NOT #"Hand aktiv" THEN #M5 := FALSE; END_IF;
   #"Tür zu" := #M5;
END_REGION

REGION Network 15: Tür auf
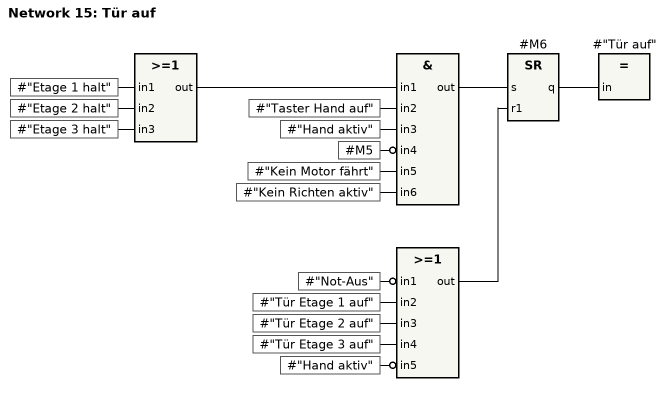
   IF (#"Etage 1 halt" OR #"Etage 2 halt" OR #"Etage 3 halt") AND #"Taster Hand auf" AND #"Hand aktiv" AND NOT #M5 AND #"Kein Motor fährt" AND #"Kein Richten aktiv" THEN
       #M6 := TRUE;   // SR flip-flop
   END_IF;
   IF NOT #"Not-Aus" OR #"Tür Etage 1 auf" OR #"Tür Etage 2 auf" OR #"Tür Etage 3 auf" OR NOT #"Hand aktiv" THEN
       #M6 := FALSE;
   END_IF;
   #"Tür auf" := #M6;
END_REGION
END_FUNCTION_BLOCK